LIN {X 0,Y 255.439,Z 401.538,A -85,B 0,C 180,E1 -18832.437,E2 -18832.437} C_VEL
LIN {X 0,Y 256.789,Z 390.953,A -85,B 0,C 180,E1 -18833.483,E2 -18833.483} C_VEL
LIN {X 0,Y 258.093,Z 377.272,A -85,B 0,C 180,E1 -18834.477,E2 -18834.477} C_VEL
LIN {X 0,Y 258.954,Z 364.44,A -85,B 0,C 180,E1 -18835.086,E2 -18835.086} C_VEL
LIN {X 0,Y 260.512,Z 307.195,A -85,B 0,C 180,E1 -18836.666,E2 -18836.666} C_VEL
LIN {X 0,Y 255.164,Z 263.56,A -85,B 0,C 180,E1 -18838.451,E2 -18838.451} C_VEL
LIN {X 0,Y 252.783,Z 256.222,A -85,B 0,C 180,E1 -18838.949,E2 -18838.949} C_VEL
LIN {X 0,Y 250.577,Z 245.438,A -85,B 0,C 180,E1 -18842.709,E2 -18842.709} C_VEL
LIN {X 0,Y 249.091,Z 238.46,A -85,B 0,C 180,E1 -18845.287,E2 -18845.287} C_VEL
LIN {X 0,Y 249.013,Z 238.47,A -85,B 0,C 180,E1 -18848.375,E2 -18848.375} C_VEL
LIN {X 0,Y 248.994,Z 238.467,A -85,B 0,C 180,E1 -18852.788,E2 -18852.788} C_VEL
LIN {X 0,Y 249.037,Z 238.464,A -85,B 0,C 180,E1 -18857.367,E2 -18857.367} C_VEL
LIN {X 0,Y 249.028,Z 238.466,A -85,B 0,C 180,E1 -18861.619,E2 -18861.619} C_VEL
LIN {X 0,Y 249.021,Z 238.467,A -85,B 0,C 180,E1 -18865.635,E2 -18865.635} C_VEL
LIN {X 0,Y 249.024,Z 238.466,A -85,B 0,C 180,E1 -18869.469,E2 -18869.469} C_VEL
LIN {X 0,Y 249.046,Z 238.462,A -85,B 0,C 180,E1 -18873.158,E2 -18873.158} C_VEL
LIN {X 0,Y 249.059,Z 238.457,A -85,B 0,C 180,E1 -18876.73,E2 -18876.73} C_VEL
LIN {X 0,Y 249.112,Z 238.451,A -85,B 0,C 180,E1 -18880.211,E2 -18880.211} C_VEL
LIN {X 0,Y 249.164,Z 238.448,A -85,B 0,C 180,E1 -18883.616,E2 -18883.616} C_VEL
LIN {X 0,Y 249.208,Z 238.435,A -85,B 0,C 180,E1 -18888.614,E2 -18888.614} C_VEL
LIN {X 0,Y 249.446,Z 238.411,A -85,B 0,C 180,E1 -18891.901,E2 -18891.901} C_VEL
LIN {X 0,Y 249.393,Z 238.406,A -85,B 0,C 180,E1 -18896.769,E2 -18896.769} C_VEL
LIN {X 0,Y 249.681,Z 238.355,A -85,B 0,C 180,E1 -18899.999,E2 -18899.999} C_VEL
LIN {X 0,Y 249.388,Z 238.41,A -85,B 0,C 180,E1 -18903.231,E2 -18903.231} C_VEL
LIN {X 0,Y 249.394,Z 238.415,A -85,B 0,C 180,E1 -18906.789,E2 -18906.789} C_VEL
LIN {X 0,Y 249.299,Z 238.426,A -85,B 0,C 180,E1 -18909.738,E2 -18909.738} C_VEL
LIN {X 0,Y 249.134,Z 238.452,A -85,B 0,C 180,E1 -18914.707,E2 -18914.707} C_VEL
LIN {X 0,Y 249.059,Z 238.457,A -85,B 0,C 180,E1 -18918.083,E2 -18918.083} C_VEL
LIN {X 0,Y 249.013,Z 238.463,A -85,B 0,C 180,E1 -18921.524,E2 -18921.524} C_VEL
LIN {X 0,Y 249.082,Z 238.453,A -85,B 0,C 180,E1 -18925.476,E2 -18925.476} C_VEL
LIN {X 0,Y 249.023,Z 238.445,A -85,B 0,C 180,E1 -18928.983,E2 -18928.983} C_VEL
LIN {X 0,Y 248.998,Z 238.45,A -85,B 0,C 180,E1 -18932.43,E2 -18932.43} C_VEL
LIN {X 0,Y 249.02,Z 238.465,A -85,B 0,C 180,E1 -18936.346,E2 -18936.346} C_VEL
LIN {X 0,Y 248.967,Z 238.464,A -85,B 0,C 180,E1 -18940.485,E2 -18940.485} C_VEL
LIN {X 0,Y 248.977,Z 238.453,A -85,B 0,C 180,E1 -18942.794,E2 -18942.794} C_VEL
LIN {X 0,Y 248.988,Z 238.468,A -85,B 0,C 180,E1 -18947.366,E2 -18947.366} C_VEL
LIN {X 0,Y 249.025,Z 238.455,A -85,B 0,C 180,E1 -18952.205,E2 -18952.205} C_VEL
LIN {X 0,Y 249.028,Z 238.464,A -85,B 0,C 180,E1 -18955.644,E2 -18955.644} C_VEL
LIN {X 0,Y 249.033,Z 238.457,A -85,B 0,C 180,E1 -18959.477,E2 -18959.477} C_VEL
LIN {X 0,Y 249.056,Z 238.46,A -85,B 0,C 180,E1 -18963.166,E2 -18963.166} C_VEL
LIN {X 0,Y 249.05,Z 238.461,A -85,B 0,C 180,E1 -18966.735,E2 -18966.735} C_VEL
LIN {X 0,Y 249.073,Z 238.462,A -85,B 0,C 180,E1 -18970.213,E2 -18970.213} C_VEL
LIN {X 0,Y 249.189,Z 238.45,A -85,B 0,C 180,E1 -18973.623,E2 -18973.623} C_VEL
LIN {X 0,Y 249.19,Z 238.451,A -85,B 0,C 180,E1 -18975.908,E2 -18975.908} C_VEL
LIN {X 0,Y 250.326,Z 241.478,A -85,B 0,C 180,E1 -18976.126,E2 -18976.126} C_VEL
LIN {X 0,Y 257.039,Z 256.974,A -85,B 0,C 180,E1 -18977.261,E2 -18977.261} C_VEL
LIN {X 0,Y 261.575,Z 270.407,A -85,B 0,C 180,E1 -18978.077,E2 -18978.077} C_VEL
LIN {X 0,Y 259.215,Z 342.899,A -85,B 0,C 180,E1 -18980.048,E2 -18980.048} C_VEL
LIN {X 0,Y 258.535,Z 356.06,A -85,B 0,C 180,E1 -18980.715,E2 -18980.715} C_VEL
LIN {X 0,Y 257.47,Z 368.762,A -85,B 0,C 180,E1 -18981.666,E2 -18981.666} C_VEL
LIN {X 0,Y 256.168,Z 380.863,A -85,B 0,C 180,E1 -18982.912,E2 -18982.912} C_VEL
LIN {X 0,Y 254.83,Z 392.116,A -85,B 0,C 180,E1 -18984.429,E2 -18984.429} C_VEL
LIN {X 0,Y 253.272,Z 402.421,A -85,B 0,C 180,E1 -18986.165,E2 -18986.165} C_VEL
LIN {X 0,Y 251.828,Z 411.246,A -85,B 0,C 180,E1 -18988.004,E2 -18988.004} C_VEL
LIN {X 0,Y 250.326,Z 420.436,A -85,B 0,C 180,E1 -18990.405,E2 -18990.405} C_VEL
LIN {X 0,Y 249.109,Z 427.844,A -85,B 0,C 180,E1 -18992.832,E2 -18992.832} C_VEL
LIN {X 0,Y 248.344,Z 432.864,A -85,B 0,C 180,E1 -18994.873,E2 -18994.873} C_VEL
LIN {X 0,Y 247.817,Z 437.113,A -85,B 0,C 180,E1 -18996.985,E2 -18996.985} C_VEL
LIN {X 0,Y 247.217,Z 441.489,A -85,B 0,C 180,E1 -18999.823,E2 -18999.823} C_VEL
LIN {X 0,Y 246.964,Z 443.438,A -85,B 0,C 180,E1 -19001.492,E2 -19001.492} C_VEL
LIN {X 0,Y 246.843,Z 445.788,A -85,B 0,C 180,E1 -19004.528,E2 -19004.528} C_VEL
LIN {X 0,Y 246.862,Z 446.599,A -85,B 0,C 180,E1 -19006.542,E2 -19006.542} C_VEL
LIN {X 0,Y 247.056,Z 446.823,A -85,B 0,C 180,E1 -19008.236,E2 -19008.236} C_VEL
LIN {X 0,Y 247.456,Z 446.467,A -85,B 0,C 180,E1 -19010.41,E2 -19010.41} C_VEL
LIN {X 0,Y 248.319,Z 444.912,A -85,B 0,C 180,E1 -19013.344,E2 -19013.344} C_VEL
LIN {X 0,Y 249.244,Z 442.844,A -85,B 0,C 180,E1 -19015.537,E2 -19015.537} C_VEL
LIN {X 0,Y 250.877,Z 438.906,A -85,B 0,C 180,E1 -19018.44,E2 -19018.44} C_VEL
LIN {X 0,Y 252.748,Z 434.14,A -85,B 0,C 180,E1 -19020.958,E2 -19020.958} C_VEL
LIN {X 0,Y 254.976,Z 427.989,A -85,B 0,C 180,E1 -19023.454,E2 -19023.454} C_VEL
LIN {X 0,Y 257.689,Z 420.236,A -85,B 0,C 180,E1 -19025.9,E2 -19025.9} C_VEL
LIN {X 0,Y 260.217,Z 412.22,A -85,B 0,C 180,E1 -19027.91,E2 -19027.91} C_VEL
LIN {X 0,Y 263.021,Z 402.281,A -85,B 0,C 180,E1 -19029.887,E2 -19029.887} C_VEL
LIN {X 0,Y 265.849,Z 391.372,A -85,B 0,C 180,E1 -19031.58,E2 -19031.58} C_VEL
LIN {X 0,Y 268.172,Z 380.195,A -85,B 0,C 180,E1 -19032.951,E2 -19032.951} C_VEL
LIN {X 0,Y 270.145,Z 367.926,A -85,B 0,C 180,E1 -19034.099,E2 -19034.099} C_VEL
LIN {X 0,Y 271.693,Z 355.388,A -85,B 0,C 180,E1 -19034.95,E2 -19034.95} C_VEL
LIN {X 0,Y 272.704,Z 342.7,A -85,B 0,C 180,E1 -19035.523,E2 -19035.523} C_VEL
LIN {X 0,Y 275.249,Z 284.695,A -85,B 0,C 180,E1 -19037.046,E2 -19037.046} C_VEL
LIN {X 0,Y 268.843,Z 271.231,A -85,B 0,C 180,E1 -19038.57,E2 -19038.57} C_VEL
LIN {X 0,Y 262.355,Z 259.216,A -85,B 0,C 180,E1 -19040.176,E2 -19040.176} C_VEL
LIN {X 0,Y 256.72,Z 250.714,A -85,B 0,C 180,E1 -19041.604,E2 -19041.604} C_VEL
LIN {X 0,Y 254.038,Z 246.769,A -85,B 0,C 180,E1 -19042.316,E2 -19042.316} C_VEL
LIN {X 0,Y 251.753,Z 243.157,A -85,B 0,C 180,E1 -19042.95,E2 -19042.95} C_VEL
LIN {X 0,Y 249.857,Z 240.911,A -85,B 0,C 180,E1 -19043.461,E2 -19043.461} C_VEL
LIN {X 0,Y 249.066,Z 238.461,A -85,B 0,C 180,E1 -19043.749,E2 -19043.749} C_VEL
LIN {X 0,Y 249.03,Z 238.456,A -85,B 0,C 180,E1 -19047.845,E2 -19047.845} C_VEL
LIN {X 0,Y 249.077,Z 238.447,A -85,B 0,C 180,E1 -19051.336,E2 -19051.336} C_VEL
LIN {X 0,Y 249.142,Z 238.437,A -85,B 0,C 180,E1 -19054.968,E2 -19054.968} C_VEL
LIN {X 0,Y 249.099,Z 238.45,A -85,B 0,C 180,E1 -19060.211,E2 -19060.211} C_VEL
LIN {X 0,Y 249.194,Z 238.434,A -85,B 0,C 180,E1 -19063.619,E2 -19063.619} C_VEL
LIN {X 0,Y 249.222,Z 238.435,A -85,B 0,C 180,E1 -19068.616,E2 -19068.616} C_VEL
LIN {X 0,Y 249.434,Z 238.4,A -85,B 0,C 180,E1 -19071.902,E2 -19071.902} C_VEL
LIN {X 0,Y 249.272,Z 238.426,A -85,B 0,C 180,E1 -19075.149,E2 -19075.149} C_VEL
LIN {X 0,Y 249.658,Z 238.38,A -85,B 0,C 180,E1 -19078.387,E2 -19078.387} C_VEL
LIN {X 0,Y 249.65,Z 238.369,A -85,B 0,C 180,E1 -19081.322,E2 -19081.322} C_VEL
LIN {X 0,Y 248.99,Z 238.46,A -85,B 0,C 180,E1 -19082.664,E2 -19082.664} C_VEL
LIN {X 0,Y 246.087,Z 238.832,A -85,B 0,C 180,E1 -19084.85,E2 -19084.85} C_VEL
LIN {X 0,Y 243.578,Z 239.148,A -85,B 0,C 180,E1 -19086.631,E2 -19086.631} C_VEL
LIN {X 0,Y 242.459,Z 239.28,A -85,B 0,C 180,E1 -19088.014,E2 -19088.014} C_VEL
LIN {X 0,Y 242.346,Z 239.289,A -85,B 0,C 180,E1 -19088.484,E2 -19088.484} C_VEL
LIN {X 0,Y 242.12,Z 239.317,A -85,B 0,C 180,E1 -19093.428,E2 -19093.428} C_VEL
LIN {X 0,Y 242.093,Z 239.326,A -85,B 0,C 180,E1 -19096.877,E2 -19096.877} C_VEL
LIN {X 0,Y 241.972,Z 239.339,A -85,B 0,C 180,E1 -19102.184,E2 -19102.184} C_VEL
LIN {X 0,Y 242.026,Z 239.337,A -85,B 0,C 180,E1 -19105.822,E2 -19105.822} C_VEL
LIN {X 0,Y 241.96,Z 239.346,A -85,B 0,C 180,E1 -19109.59,E2 -19109.59} C_VEL
LIN {X 0,Y 241.963,Z 239.342,A -85,B 0,C 180,E1 -19113.496,E2 -19113.496} C_VEL
LIN {X 0,Y 241.98,Z 239.336,A -85,B 0,C 180,E1 -19117.584,E2 -19117.584} C_VEL
LIN {X 0,Y 241.924,Z 239.326,A -85,B 0,C 180,E1 -19121.926,E2 -19121.926} C_VEL
LIN {X 0,Y 241.981,Z 239.548,A -85,B 0,C 180,E1 -19123.291,E2 -19123.291} C_VEL
LIN {X 0,Y 244.202,Z 246.816,A -85,B 0,C 180,E1 -19127.212,E2 -19127.212} C_VEL
LIN {X 0,Y 246.291,Z 254.002,A -85,B 0,C 180,E1 -19130.671,E2 -19130.671} C_VEL
LIN {X 0,Y 249.147,Z 258.875,A -85,B 0,C 180,E1 -19131.514,E2 -19131.514} C_VEL
LIN {X 0,Y 255.372,Z 270.327,A -85,B 0,C 180,E1 -19133.278,E2 -19133.278} C_VEL
LIN {X 0,Y 261.811,Z 283.473,A -85,B 0,C 180,E1 -19135.011,E2 -19135.011} C_VEL
LIN {X 0,Y 265.059,Z 291.167,A -85,B 0,C 180,E1 -19135.87,E2 -19135.87} C_VEL
LIN {X 0,Y 268.477,Z 313.345,A -85,B 0,C 180,E1 -19137.216,E2 -19137.216} C_VEL
LIN {X 0,Y 266.163,Z 364.461,A -85,B 0,C 180,E1 -19138.609,E2 -19138.609} C_VEL
LIN {X 0,Y 264.74,Z 377.806,A -85,B 0,C 180,E1 -19139.228,E2 -19139.228} C_VEL
LIN {X 0,Y 262.748,Z 390.649,A -85,B 0,C 180,E1 -19140.12,E2 -19140.12} C_VEL
LIN {X 0,Y 260.478,Z 401.692,A -85,B 0,C 180,E1 -19141.165,E2 -19141.165} C_VEL
LIN {X 0,Y 257.609,Z 413.215,A -85,B 0,C 180,E1 -19142.588,E2 -19142.588} C_VEL
LIN {X 0,Y 254.685,Z 423.609,A -85,B 0,C 180,E1 -19144.238,E2 -19144.238} C_VEL
LIN {X 0,Y 251.769,Z 433.003,A -85,B 0,C 180,E1 -19146.123,E2 -19146.123} C_VEL
LIN {X 0,Y 248.699,Z 442.088,A -85,B 0,C 180,E1 -19148.446,E2 -19148.446} C_VEL
LIN {X 0,Y 246.223,Z 449.442,A -85,B 0,C 180,E1 -19150.836,E2 -19150.836} C_VEL
LIN {X 0,Y 244.09,Z 455.377,A -85,B 0,C 180,E1 -19153.265,E2 -19153.265} C_VEL
LIN {X 0,Y 242.298,Z 460.092,A -85,B 0,C 180,E1 -19155.725,E2 -19155.725} C_VEL
LIN {X 0,Y 241.137,Z 463.725,A -85,B 0,C 180,E1 -19158.226,E2 -19158.226} C_VEL
LIN {X 0,Y 240.576,Z 465.619,A -85,B 0,C 180,E1 -19159.903,E2 -19159.903} C_VEL
LIN {X 0,Y 239.903,Z 468.104,A -85,B 0,C 180,E1 -19163.268,E2 -19163.268} C_VEL
LIN {X 0,Y 239.849,Z 468.8,A -85,B 0,C 180,E1 -19165.049,E2 -19165.049} C_VEL
LIN {X 0,Y 239.881,Z 469.054,A -85,B 0,C 180,E1 -19166.638,E2 -19166.638} C_VEL
LIN {X 0,Y 239.976,Z 468.912,A -85,B 0,C 180,E1 -19168.319,E2 -19168.319} C_VEL
LIN {X 0,Y 240.024,Z 468.36,A -85,B 0,C 180,E1 -19169.997,E2 -19169.997} C_VEL
LIN {X 0,Y 240.008,Z 467.408,A -85,B 0,C 180,E1 -19171.675,E2 -19171.675} C_VEL
LIN {X 0,Y 239.963,Z 466.048,A -85,B 0,C 180,E1 -19173.355,E2 -19173.355} C_VEL
LIN {X 0,Y 239.964,Z 463.14,A -85,B 0,C 180,E1 -19175.879,E2 -19175.879} C_VEL
LIN {X 0,Y 240.191,Z 459.169,A -85,B 0,C 180,E1 -19178.409,E2 -19178.409} C_VEL
LIN {X 0,Y 240.757,Z 453.024,A -85,B 0,C 180,E1 -19181.36,E2 -19181.36} C_VEL
LIN {X 0,Y 241.717,Z 446.284,A -85,B 0,C 180,E1 -19183.875,E2 -19183.875} C_VEL
LIN {X 0,Y 243.073,Z 437.902,A -85,B 0,C 180,E1 -19186.369,E2 -19186.369} C_VEL
LIN {X 0,Y 244.393,Z 429.258,A -85,B 0,C 180,E1 -19188.436,E2 -19188.436} C_VEL
LIN {X 0,Y 245.963,Z 419.772,A -85,B 0,C 180,E1 -19190.266,E2 -19190.266} C_VEL
LIN {X 0,Y 247.529,Z 409.43,A -85,B 0,C 180,E1 -19191.874,E2 -19191.874} C_VEL
LIN {X 0,Y 249.152,Z 398.134,A -85,B 0,C 180,E1 -19193.255,E2 -19193.255} C_VEL
LIN {X 0,Y 250.64,Z 385.426,A -85,B 0,C 180,E1 -19194.425,E2 -19194.425} C_VEL
LIN {X 0,Y 251.846,Z 371.806,A -85,B 0,C 180,E1 -19195.291,E2 -19195.291} C_VEL
LIN {X 0,Y 252.465,Z 359.698,A -85,B 0,C 180,E1 -19195.777,E2 -19195.777} C_VEL
LIN {X 0,Y 253.92,Z 308.786,A -85,B 0,C 180,E1 -19197.194,E2 -19197.194} C_VEL
LIN {X 0,Y 248.987,Z 266.806,A -85,B 0,C 180,E1 -19198.952,E2 -19198.952} C_VEL
LIN {X 0,Y 247.974,Z 262.879,A -85,B 0,C 180,E1 -19199.176,E2 -19199.176} C_VEL
LIN {X 0,Y 245.566,Z 256.004,A -85,B 0,C 180,E1 -19199.648,E2 -19199.648} C_VEL
LIN {X 0,Y 243.171,Z 244.542,A -85,B 0,C 180,E1 -19203.797,E2 -19203.797} C_VEL
LIN {X 0,Y 242.034,Z 239.342,A -85,B 0,C 180,E1 -19205.796,E2 -19205.796} C_VEL
LIN {X 0,Y 241.941,Z 239.35,A -85,B 0,C 180,E1 -19209.714,E2 -19209.714} C_VEL
LIN {X 0,Y 241.919,Z 239.35,A -85,B 0,C 180,E1 -19214.196,E2 -19214.196} C_VEL
LIN {X 0,Y 241.961,Z 239.346,A -85,B 0,C 180,E1 -19218.082,E2 -19218.082} C_VEL
LIN {X 0,Y 241.985,Z 239.34,A -85,B 0,C 180,E1 -19222.417,E2 -19222.417} C_VEL
LIN {X 0,Y 241.957,Z 239.342,A -85,B 0,C 180,E1 -19226.503,E2 -19226.503} C_VEL
LIN {X 0,Y 242.01,Z 239.335,A -85,B 0,C 180,E1 -19230.584,E2 -19230.584} C_VEL
LIN {X 0,Y 242.04,Z 239.333,A -85,B 0,C 180,E1 -19234.179,E2 -19234.179} C_VEL
LIN {X 0,Y 242.055,Z 239.332,A -85,B 0,C 180,E1 -19238.275,E2 -19238.275} C_VEL
LIN {X 0,Y 242.124,Z 239.323,A -85,B 0,C 180,E1 -19243.282,E2 -19243.282} C_VEL
LIN {X 0,Y 242.139,Z 239.315,A -85,B 0,C 180,E1 -19248.277,E2 -19248.277} C_VEL
LIN {X 0,Y 242.393,Z 239.291,A -85,B 0,C 180,E1 -19251.664,E2 -19251.664} C_VEL
LIN {X 0,Y 242.219,Z 239.307,A -85,B 0,C 180,E1 -19255.006,E2 -19255.006} C_VEL
LIN {X 0,Y 242.597,Z 239.242,A -85,B 0,C 180,E1 -19258.339,E2 -19258.339} C_VEL
LIN {X 0,Y 242.595,Z 239.247,A -85,B 0,C 180,E1 -19261.66,E2 -19261.66} C_VEL
LIN {X 0,Y 242.373,Z 239.292,A -85,B 0,C 180,E1 -19266.762,E2 -19266.762} C_VEL
LIN {X 0,Y 242.228,Z 239.306,A -85,B 0,C 180,E1 -19270.025,E2 -19270.025} C_VEL
LIN {X 0,Y 242.086,Z 239.33,A -85,B 0,C 180,E1 -19275.145,E2 -19275.145} C_VEL
LIN {X 0,Y 241.996,Z 239.335,A -85,B 0,C 180,E1 -19278.63,E2 -19278.63} C_VEL
LIN {X 0,Y 241.956,Z 239.343,A -85,B 0,C 180,E1 -19282.185,E2 -19282.185} C_VEL
LIN {X 0,Y 242.02,Z 239.333,A -85,B 0,C 180,E1 -19285.832,E2 -19285.832} C_VEL
LIN {X 0,Y 241.946,Z 239.324,A -85,B 0,C 180,E1 -19289.591,E2 -19289.591} C_VEL
LIN {X 0,Y 241.951,Z 239.335,A -85,B 0,C 180,E1 -19293.497,E2 -19293.497} C_VEL
LIN {X 0,Y 241.962,Z 239.342,A -85,B 0,C 180,E1 -19297.586,E2 -19297.586} C_VEL
LIN {X 0,Y 241.906,Z 239.337,A -85,B 0,C 180,E1 -19301.928,E2 -19301.928} C_VEL
LIN {X 0,Y 241.904,Z 239.352,A -85,B 0,C 180,E1 -19306.578,E2 -19306.578} C_VEL
LIN {X 0,Y 241.977,Z 239.334,A -85,B 0,C 180,E1 -19311.645,E2 -19311.645} C_VEL
LIN {X 0,Y 241.964,Z 239.343,A -85,B 0,C 180,E1 -19314.493,E2 -19314.493} C_VEL
LIN {X 0,Y 241.958,Z 239.339,A -85,B 0,C 180,E1 -19318.484,E2 -19318.484} C_VEL
LIN {X 0,Y 241.989,Z 239.343,A -85,B 0,C 180,E1 -19322.316,E2 -19322.316} C_VEL
LIN {X 0,Y 242.03,Z 239.337,A -85,B 0,C 180,E1 -19326.019,E2 -19326.019} C_VEL
LIN {X 0,Y 242.01,Z 239.341,A -85,B 0,C 180,E1 -19329.611,E2 -19329.611} C_VEL
LIN {X 0,Y 242.109,Z 239.332,A -85,B 0,C 180,E1 -19333.32,E2 -19333.32} C_VEL
LIN {X 0,Y 242.154,Z 239.407,A -85,B 0,C 180,E1 -19335.201,E2 -19335.201} C_VEL
LIN {X 0,Y 243.167,Z 242.232,A -85,B 0,C 180,E1 -19335.402,E2 -19335.402} C_VEL
LIN {X 0,Y 250.184,Z 257.809,A -85,B 0,C 180,E1 -19336.62,E2 -19336.62} C_VEL
LIN {X 0,Y 254.989,Z 271.769,A -85,B 0,C 180,E1 -19337.515,E2 -19337.515} C_VEL
LIN {X 0,Y 252.534,Z 343.875,A -85,B 0,C 180,E1 -19339.531,E2 -19339.531} C_VEL
LIN {X 0,Y 251.772,Z 357.541,A -85,B 0,C 180,E1 -19340.261,E2 -19340.261} C_VEL
LIN {X 0,Y 250.666,Z 369.927,A -85,B 0,C 180,E1 -19341.235,E2 -19341.235} C_VEL
LIN {X 0,Y 249.317,Z 381.794,A -85,B 0,C 180,E1 -19342.512,E2 -19342.512} C_VEL
LIN {X 0,Y 247.812,Z 393.628,A -85,B 0,C 180,E1 -19344.175,E2 -19344.175} C_VEL
LIN {X 0,Y 246.155,Z 404.168,A -85,B 0,C 180,E1 -19346.054,E2 -19346.054} C_VEL
LIN {X 0,Y 244.419,Z 414.357,A -85,B 0,C 180,E1 -19348.355,E2 -19348.355} C_VEL
LIN {X 0,Y 243.176,Z 421.706,A -85,B 0,C 180,E1 -19350.417,E2 -19350.417} C_VEL
LIN {X 0,Y 241.98,Z 428.94,A -85,B 0,C 180,E1 -19352.916,E2 -19352.916} C_VEL
LIN {X 0,Y 241.206,Z 433.823,A -85,B 0,C 180,E1 -19355.017,E2 -19355.017} C_VEL
LIN {X 0,Y 240.569,Z 438.563,A -85,B 0,C 180,E1 -19357.556,E2 -19357.556} C_VEL
LIN {X 0,Y 240.056,Z 442.199,A -85,B 0,C 180,E1 -19360.119,E2 -19360.119} C_VEL
LIN {X 0,Y 239.843,Z 444.046,A -85,B 0,C 180,E1 -19361.838,E2 -19361.838} C_VEL
LIN {X 0,Y 239.753,Z 446.126,A -85,B 0,C 180,E1 -19364.685,E2 -19364.685} C_VEL
LIN {X 0,Y 239.821,Z 447.01,A -85,B 0,C 180,E1 -19367.042,E2 -19367.042} C_VEL
LIN {X 0,Y 240.053,Z 447.131,A -85,B 0,C 180,E1 -19368.788,E2 -19368.788} C_VEL
LIN {X 0,Y 240.439,Z 446.8,A -85,B 0,C 180,E1 -19370.716,E2 -19370.716} C_VEL
LIN {X 0,Y 240.88,Z 446.156,A -85,B 0,C 180,E1 -19372.291,E2 -19372.291} C_VEL
LIN {X 0,Y 241.471,Z 444.998,A -85,B 0,C 180,E1 -19374.047,E2 -19374.047} C_VEL
LIN {X 0,Y 242.342,Z 443.2,A -85,B 0,C 180,E1 -19375.973,E2 -19375.973} C_VEL
LIN {X 0,Y 243.732,Z 440.081,A -85,B 0,C 180,E1 -19378.41,E2 -19378.41} C_VEL
LIN {X 0,Y 245.62,Z 435.601,A -85,B 0,C 180,E1 -19381,E2 -19381} C_VEL
LIN {X 0,Y 247.883,Z 429.807,A -85,B 0,C 180,E1 -19383.564,E2 -19383.564} C_VEL
LIN {X 0,Y 250.653,Z 422.421,A -85,B 0,C 180,E1 -19386.073,E2 -19386.073} C_VEL
LIN {X 0,Y 253.201,Z 414.791,A -85,B 0,C 180,E1 -19388.139,E2 -19388.139} C_VEL
LIN {X 0,Y 256.282,Z 404.734,A -85,B 0,C 180,E1 -19390.303,E2 -19390.303} C_VEL
LIN {X 0,Y 259.021,Z 395.064,A -85,B 0,C 180,E1 -19391.923,E2 -19391.923} C_VEL
LIN {X 0,Y 261.61,Z 383.714,A -85,B 0,C 180,E1 -19393.436,E2 -19393.436} C_VEL
LIN {X 0,Y 263.736,Z 371.991,A -85,B 0,C 180,E1 -19394.653,E2 -19394.653} C_VEL
LIN {X 0,Y 265.523,Z 359.394,A -85,B 0,C 180,E1 -19395.613,E2 -19395.613} C_VEL
LIN {X 0,Y 266.799,Z 346.003,A -85,B 0,C 180,E1 -19396.297,E2 -19396.297} C_VEL
LIN {X 0,Y 268.025,Z 322.583,A -85,B 0,C 180,E1 -19396.962,E2 -19396.962} C_VEL
LIN {X 0,Y 269.62,Z 286.994,A -85,B 0,C 180,E1 -19397.899,E2 -19397.899} C_VEL
LIN {X 0,Y 262.712,Z 272.581,A -85,B 0,C 180,E1 -19399.628,E2 -19399.628} C_VEL
LIN {X 0,Y 256.927,Z 262.324,A -85,B 0,C 180,E1 -19401.124,E2 -19401.124} C_VEL
LIN {X 0,Y 250.399,Z 252.33,A -85,B 0,C 180,E1 -19402.884,E2 -19402.884} C_VEL
LIN {X 0,Y 247.34,Z 247.994,A -85,B 0,C 180,E1 -19403.746,E2 -19403.746} C_VEL
LIN {X 0,Y 245.179,Z 244.537,A -85,B 0,C 180,E1 -19404.395,E2 -19404.395} C_VEL
LIN {X 0,Y 242.833,Z 241.862,A -85,B 0,C 180,E1 -19405.076,E2 -19405.076} C_VEL
LIN {X 0,Y 242.014,Z 239.331,A -85,B 0,C 180,E1 -19405.415,E2 -19405.415} C_VEL
LIN {X 0,Y 241.999,Z 239.334,A -85,B 0,C 180,E1 -19410.416,E2 -19410.416} C_VEL
LIN {X 0,Y 242.06,Z 239.323,A -85,B 0,C 180,E1 -19414.183,E2 -19414.183} C_VEL
LIN {X 0,Y 242.044,Z 239.323,A -85,B 0,C 180,E1 -19418.298,E2 -19418.298} C_VEL
LIN {X 0,Y 242.154,Z 239.309,A -85,B 0,C 180,E1 -19423.278,E2 -19423.278} C_VEL
LIN {X 0,Y 242.157,Z 239.312,A -85,B 0,C 180,E1 -19428.279,E2 -19428.279} C_VEL
LIN {X 0,Y 242.381,Z 239.279,A -85,B 0,C 180,E1 -19431.665,E2 -19431.665} C_VEL
LIN {X 0,Y 242.405,Z 239.282,A -85,B 0,C 180,E1 -19433.341,E2 -19433.341} C_VEL
LIN {X 0,Y 242.619,Z 239.257,A -85,B 0,C 180,E1 -19438.341,E2 -19438.341} C_VEL
LIN {X 0,Y 242.618,Z 239.246,A -85,B 0,C 180,E1 -19441.66,E2 -19441.66} C_VEL
LIN {X 0,Y 242.385,Z 239.276,A -85,B 0,C 180,E1 -19446.661,E2 -19446.661} C_VEL
LIN {X 0,Y 242.346,Z 239.289,A -85,B 0,C 180,E1 -19448.484,E2 -19448.484} C_VEL
LIN {X 0,Y 241.606,Z 239.374,A -85,B 0,C 180,E1 -19449.868,E2 -19449.868} C_VEL
LIN {X 0,Y 238.682,Z 239.747,A -85,B 0,C 180,E1 -19452.123,E2 -19452.123} C_VEL
LIN {X 0,Y 236.219,Z 240.049,A -85,B 0,C 180,E1 -19453.96,E2 -19453.96} C_VEL
LIN {X 0,Y 235.146,Z 240.181,A -85,B 0,C 180,E1 -19455.388,E2 -19455.388} C_VEL
LIN {X 0,Y 235.047,Z 240.194,A -85,B 0,C 180,E1 -19455.872,E2 -19455.872} C_VEL
LIN {X 0,Y 234.93,Z 240.22,A -85,B 0,C 180,E1 -19461.038,E2 -19461.038} C_VEL
LIN {X 0,Y 234.962,Z 240.213,A -85,B 0,C 180,E1 -19466.194,E2 -19466.194} C_VEL
LIN {X 0,Y 234.883,Z 240.219,A -85,B 0,C 180,E1 -19470.575,E2 -19470.575} C_VEL
LIN {X 0,Y 234.894,Z 240.218,A -85,B 0,C 180,E1 -19474.645,E2 -19474.645} C_VEL
LIN {X 0,Y 234.91,Z 240.225,A -85,B 0,C 180,E1 -19478.936,E2 -19478.936} C_VEL
LIN {X 0,Y 234.894,Z 240.225,A -85,B 0,C 180,E1 -19481.584,E2 -19481.584} C_VEL
LIN {X 0,Y 237.287,Z 247.923,A -85,B 0,C 180,E1 -19486.02,E2 -19486.02} C_VEL
LIN {X 0,Y 238.935,Z 253.518,A -85,B 0,C 180,E1 -19488.863,E2 -19488.863} C_VEL
LIN {X 0,Y 241.712,Z 258.238,A -85,B 0,C 180,E1 -19489.762,E2 -19489.762} C_VEL
LIN {X 0,Y 246.409,Z 266.402,A -85,B 0,C 180,E1 -19491.204,E2 -19491.204} C_VEL
LIN {X 0,Y 251.242,Z 275.433,A -85,B 0,C 180,E1 -19492.619,E2 -19492.619} C_VEL
LIN {X 0,Y 257.32,Z 288.042,A -85,B 0,C 180,E1 -19494.325,E2 -19494.325} C_VEL
LIN {X 0,Y 259.874,Z 294.298,A -85,B 0,C 180,E1 -19495.039,E2 -19495.039} C_VEL
LIN {X 0,Y 262.897,Z 314.711,A -85,B 0,C 180,E1 -19496.311,E2 -19496.311} C_VEL
LIN {X 0,Y 260.482,Z 364.486,A -85,B 0,C 180,E1 -19497.686,E2 -19497.686} C_VEL
LIN {X 0,Y 258.965,Z 378.06,A -85,B 0,C 180,E1 -19498.334,E2 -19498.334} C_VEL
LIN {X 0,Y 257.054,Z 389.808,A -85,B 0,C 180,E1 -19499.16,E2 -19499.16} C_VEL
LIN {X 0,Y 254.693,Z 400.991,A -85,B 0,C 180,E1 -19500.218,E2 -19500.218} C_VEL
LIN {X 0,Y 251.697,Z 412.585,A -85,B 0,C 180,E1 -19501.661,E2 -19501.661} C_VEL
LIN {X 0,Y 248.623,Z 423.031,A -85,B 0,C 180,E1 -19503.336,E2 -19503.336} C_VEL
LIN {X 0,Y 245.876,Z 431.591,A -85,B 0,C 180,E1 -19505.063,E2 -19505.063} C_VEL
LIN {X 0,Y 243.106,Z 439.509,A -85,B 0,C 180,E1 -19507.028,E2 -19507.028} C_VEL
LIN {X 0,Y 240.321,Z 447.298,A -85,B 0,C 180,E1 -19509.455,E2 -19509.455} C_VEL
LIN {X 0,Y 237.945,Z 453.566,A -85,B 0,C 180,E1 -19511.932,E2 -19511.932} C_VEL
LIN {X 0,Y 235.983,Z 458.587,A -85,B 0,C 180,E1 -19514.451,E2 -19514.451} C_VEL
LIN {X 0,Y 234.473,Z 462.505,A -85,B 0,C 180,E1 -19517.007,E2 -19517.007} C_VEL
LIN {X 0,Y 233.555,Z 465.429,A -85,B 0,C 180,E1 -19519.596,E2 -19519.596} C_VEL
LIN {X 0,Y 232.824,Z 467.848,A -85,B 0,C 180,E1 -19523.063,E2 -19523.063} C_VEL
LIN {X 0,Y 232.775,Z 468.566,A -85,B 0,C 180,E1 -19525.107,E2 -19525.107} C_VEL
LIN {X 0,Y 232.903,Z 468.54,A -85,B 0,C 180,E1 -19528.268,E2 -19528.268} C_VEL
LIN {X 0,Y 232.952,Z 467.96,A -85,B 0,C 180,E1 -19529.997,E2 -19529.997} C_VEL
LIN {X 0,Y 232.937,Z 466.979,A -85,B 0,C 180,E1 -19531.726,E2 -19531.726} C_VEL
LIN {X 0,Y 232.879,Z 465.575,A -85,B 0,C 180,E1 -19533.457,E2 -19533.457} C_VEL
LIN {X 0,Y 232.9,Z 462.612,A -85,B 0,C 180,E1 -19536.059,E2 -19536.059} C_VEL
LIN {X 0,Y 233.127,Z 458.573,A -85,B 0,C 180,E1 -19538.666,E2 -19538.666} C_VEL
LIN {X 0,Y 233.748,Z 452.322,A -85,B 0,C 180,E1 -19541.705,E2 -19541.705} C_VEL
LIN {X 0,Y 234.788,Z 445.5,A -85,B 0,C 180,E1 -19544.293,E2 -19544.293} C_VEL
LIN {X 0,Y 236.245,Z 437.008,A -85,B 0,C 180,E1 -19546.856,E2 -19546.856} C_VEL
LIN {X 0,Y 237.623,Z 428.208,A -85,B 0,C 180,E1 -19548.981,E2 -19548.981} C_VEL
LIN {X 0,Y 239.208,Z 418.564,A -85,B 0,C 180,E1 -19550.864,E2 -19550.864} C_VEL
LIN {X 0,Y 240.837,Z 408.031,A -85,B 0,C 180,E1 -19552.515,E2 -19552.515} C_VEL
LIN {X 0,Y 242.656,Z 396.499,A -85,B 0,C 180,E1 -19553.916,E2 -19553.916} C_VEL
LIN {X 0,Y 244.035,Z 384.492,A -85,B 0,C 180,E1 -19555.018,E2 -19555.018} C_VEL
LIN {X 0,Y 245.202,Z 371.54,A -85,B 0,C 180,E1 -19555.856,E2 -19555.856} C_VEL
LIN {X 0,Y 245.908,Z 357.828,A -85,B 0,C 180,E1 -19556.403,E2 -19556.403} C_VEL
LIN {X 0,Y 247.278,Z 308.652,A -85,B 0,C 180,E1 -19557.81,E2 -19557.81} C_VEL
LIN {X 0,Y 242.457,Z 267.665,A -85,B 0,C 180,E1 -19559.587,E2 -19559.587} C_VEL
LIN {X 0,Y 238.266,Z 255.572,A -85,B 0,C 180,E1 -19560.463,E2 -19560.463} C_VEL
LIN {X 0,Y 235.704,Z 243.521,A -85,B 0,C 180,E1 -19565.013,E2 -19565.013} C_VEL
LIN {X 0,Y 234.984,Z 240.219,A -85,B 0,C 180,E1 -19566.366,E2 -19566.366} C_VEL
LIN {X 0,Y 234.928,Z 240.224,A -85,B 0,C 180,E1 -19568.939,E2 -19568.939} C_VEL
LIN {X 0,Y 234.873,Z 240.228,A -85,B 0,C 180,E1 -19573.48,E2 -19573.48} C_VEL
LIN {X 0,Y 234.941,Z 240.219,A -85,B 0,C 180,E1 -19576.526,E2 -19576.526} C_VEL
LIN {X 0,Y 234.934,Z 240.218,A -85,B 0,C 180,E1 -19581.081,E2 -19581.081} C_VEL
LIN {X 0,Y 234.911,Z 240.223,A -85,B 0,C 180,E1 -19585.358,E2 -19585.358} C_VEL
LIN {X 0,Y 234.905,Z 240.225,A -85,B 0,C 180,E1 -19589.428,E2 -19589.428} C_VEL
LIN {X 0,Y 234.967,Z 240.216,A -85,B 0,C 180,E1 -19593.79,E2 -19593.79} C_VEL
LIN {X 0,Y 235.012,Z 240.211,A -85,B 0,C 180,E1 -19598.969,E2 -19598.969} C_VEL
LIN {X 0,Y 235.06,Z 240.201,A -85,B 0,C 180,E1 -19603.062,E2 -19603.062} C_VEL
LIN {X 0,Y 235.07,Z 240.196,A -85,B 0,C 180,E1 -19607.919,E2 -19607.919} C_VEL
LIN {X 0,Y 235.342,Z 240.17,A -85,B 0,C 180,E1 -19611.412,E2 -19611.412} C_VEL
LIN {X 0,Y 235.368,Z 240.166,A -85,B 0,C 180,E1 -19613.14,E2 -19613.14} C_VEL
LIN {X 0,Y 235.557,Z 240.117,A -85,B 0,C 180,E1 -19618.29,E2 -19618.29} C_VEL
LIN {X 0,Y 235.555,Z 240.123,A -85,B 0,C 180,E1 -19621.709,E2 -19621.709} C_VEL
LIN {X 0,Y 235.331,Z 240.171,A -85,B 0,C 180,E1 -19626.86,E2 -19626.86} C_VEL
LIN {X 0,Y 235.176,Z 240.185,A -85,B 0,C 180,E1 -19630.329,E2 -19630.329} C_VEL
LIN {X 0,Y 235.035,Z 240.206,A -85,B 0,C 180,E1 -19635.611,E2 -19635.611} C_VEL
LIN {X 0,Y 234.935,Z 240.212,A -85,B 0,C 180,E1 -19639.211,E2 -19639.211} C_VEL
LIN {X 0,Y 234.911,Z 240.224,A -85,B 0,C 180,E1 -19642.887,E2 -19642.887} C_VEL
LIN {X 0,Y 234.926,Z 240.213,A -85,B 0,C 180,E1 -19646.662,E2 -19646.662} C_VEL
LIN {X 0,Y 234.872,Z 240.199,A -85,B 0,C 180,E1 -19650.576,E2 -19650.576} C_VEL
LIN {X 0,Y 234.902,Z 240.218,A -85,B 0,C 180,E1 -19654.642,E2 -19654.642} C_VEL
LIN {X 0,Y 234.888,Z 240.222,A -85,B 0,C 180,E1 -19658.939,E2 -19658.939} C_VEL
LIN {X 0,Y 234.855,Z 240.21,A -85,B 0,C 180,E1 -19663.493,E2 -19663.493} C_VEL
LIN {X 0,Y 234.857,Z 240.229,A -85,B 0,C 180,E1 -19666.516,E2 -19666.516} C_VEL
LIN {X 0,Y 234.9,Z 240.216,A -85,B 0,C 180,E1 -19671.083,E2 -19671.083} C_VEL
LIN {X 0,Y 234.911,Z 240.221,A -85,B 0,C 180,E1 -19675.366,E2 -19675.366} C_VEL
LIN {X 0,Y 234.908,Z 240.215,A -85,B 0,C 180,E1 -19679.435,E2 -19679.435} C_VEL
LIN {X 0,Y 234.983,Z 240.215,A -85,B 0,C 180,E1 -19683.799,E2 -19683.799} C_VEL
LIN {X 0,Y 234.961,Z 240.217,A -85,B 0,C 180,E1 -19688.97,E2 -19688.97} C_VEL
LIN {X 0,Y 235.049,Z 240.211,A -85,B 0,C 180,E1 -19693.096,E2 -19693.096} C_VEL
LIN {X 0,Y 235.072,Z 240.209,A -85,B 0,C 180,E1 -19694.423,E2 -19694.423} C_VEL
LIN {X 0,Y 236.157,Z 243.161,A -85,B 0,C 180,E1 -19694.654,E2 -19694.654} C_VEL
LIN {X 0,Y 244.013,Z 260.374,A -85,B 0,C 180,E1 -19696.075,E2 -19696.075} C_VEL
LIN {X 0,Y 248.399,Z 273.131,A -85,B 0,C 180,E1 -19696.922,E2 -19696.922} C_VEL
LIN {X 0,Y 245.929,Z 343.671,A -85,B 0,C 180,E1 -19698.934,E2 -19698.934} C_VEL
LIN {X 0,Y 245.179,Z 356.76,A -85,B 0,C 180,E1 -19699.631,E2 -19699.631} C_VEL
LIN {X 0,Y 243.981,Z 370.004,A -85,B 0,C 180,E1 -19700.679,E2 -19700.679} C_VEL
LIN {X 0,Y 242.699,Z 381.138,A -85,B 0,C 180,E1 -19701.888,E2 -19701.888} C_VEL
LIN {X 0,Y 241.376,Z 391.399,A -85,B 0,C 180,E1 -19703.315,E2 -19703.315} C_VEL
LIN {X 0,Y 239.714,Z 402.059,A -85,B 0,C 180,E1 -19705.168,E2 -19705.168} C_VEL
LIN {X 0,Y 238.186,Z 410.787,A -85,B 0,C 180,E1 -19707.043,E2 -19707.043} C_VEL
LIN {X 0,Y 236.72,Z 418.821,A -85,B 0,C 180,E1 -19709.152,E2 -19709.152} C_VEL
LIN {X 0,Y 235.364,Z 426.671,A -85,B 0,C 180,E1 -19711.714,E2 -19711.714} C_VEL
LIN {X 0,Y 234.339,Z 432.948,A -85,B 0,C 180,E1 -19714.302,E2 -19714.302} C_VEL
LIN {X 0,Y 233.642,Z 438.01,A -85,B 0,C 180,E1 -19716.957,E2 -19716.957} C_VEL
LIN {X 0,Y 233.084,Z 441.807,A -85,B 0,C 180,E1 -19719.548,E2 -19719.548} C_VEL
LIN {X 0,Y 232.738,Z 444.634,A -85,B 0,C 180,E1 -19722.205,E2 -19722.205} C_VEL
LIN {X 0,Y 232.656,Z 446.461,A -85,B 0,C 180,E1 -19724.842,E2 -19724.842} C_VEL
LIN {X 0,Y 232.792,Z 447.378,A -85,B 0,C 180,E1 -19727.573,E2 -19727.573} C_VEL
LIN {X 0,Y 233.425,Z 447.134,A -85,B 0,C 180,E1 -19731.038,E2 -19731.038} C_VEL
LIN {X 0,Y 233.989,Z 446.319,A -85,B 0,C 180,E1 -19732.984,E2 -19732.984} C_VEL
LIN {X 0,Y 235.486,Z 443.542,A -85,B 0,C 180,E1 -19736.449,E2 -19736.449} C_VEL
LIN {X 0,Y 237.158,Z 439.977,A -85,B 0,C 180,E1 -19739.273,E2 -19739.273} C_VEL
LIN {X 0,Y 239.234,Z 435.366,A -85,B 0,C 180,E1 -19741.924,E2 -19741.924} C_VEL
LIN {X 0,Y 241.683,Z 429.382,A -85,B 0,C 180,E1 -19744.545,E2 -19744.545} C_VEL
LIN {X 0,Y 244.622,Z 421.794,A -85,B 0,C 180,E1 -19747.108,E2 -19747.108} C_VEL
LIN {X 0,Y 247.355,Z 413.981,A -85,B 0,C 180,E1 -19749.207,E2 -19749.207} C_VEL
LIN {X 0,Y 250.439,Z 404.386,A -85,B 0,C 180,E1 -19751.259,E2 -19751.259} C_VEL
LIN {X 0,Y 253.5,Z 393.562,A -85,B 0,C 180,E1 -19753.054,E2 -19753.054} C_VEL
LIN {X 0,Y 255.994,Z 382.9,A -85,B 0,C 180,E1 -19754.456,E2 -19754.456} C_VEL
LIN {X 0,Y 258.279,Z 370.47,A -85,B 0,C 180,E1 -19755.722,E2 -19755.722} C_VEL
LIN {X 0,Y 260.149,Z 356.996,A -85,B 0,C 180,E1 -19756.694,E2 -19756.694} C_VEL
LIN {X 0,Y 261.282,Z 344.726,A -85,B 0,C 180,E1 -19757.289,E2 -19757.289} C_VEL
LIN {X 0,Y 264.022,Z 289.43,A -85,B 0,C 180,E1 -19758.79,E2 -19758.79} C_VEL
LIN {X 0,Y 257.942,Z 276.58,A -85,B 0,C 180,E1 -19760.393,E2 -19760.393} C_VEL
LIN {X 0,Y 252.55,Z 266.901,A -85,B 0,C 180,E1 -19761.851,E2 -19761.851} C_VEL
LIN {X 0,Y 246.177,Z 257.11,A -85,B 0,C 180,E1 -19763.643,E2 -19763.643} C_VEL
LIN {X 0,Y 243.26,Z 252.911,A -85,B 0,C 180,E1 -19764.505,E2 -19764.505} C_VEL
LIN {X 0,Y 240.793,Z 249.306,A -85,B 0,C 180,E1 -19765.264,E2 -19765.264} C_VEL
LIN {X 0,Y 238.588,Z 246.142,A -85,B 0,C 180,E1 -19765.967,E2 -19765.967} C_VEL
LIN {X 0,Y 237.905,Z 245.147,A -85,B 0,C 180,E1 -19766.19,E2 -19766.19} C_VEL
LIN {X 0,Y 235.835,Z 242.9,A -85,B 0,C 180,E1 -19766.845,E2 -19766.845} C_VEL
LIN {X 0,Y 234.958,Z 240.212,A -85,B 0,C 180,E1 -19767.233,E2 -19767.233} C_VEL
LIN {X 0,Y 234.928,Z 240.209,A -85,B 0,C 180,E1 -19771.403,E2 -19771.403} C_VEL
LIN {X 0,Y 234.978,Z 240.201,A -85,B 0,C 180,E1 -19775.246,E2 -19775.246} C_VEL
LIN {X 0,Y 235.002,Z 240.198,A -85,B 0,C 180,E1 -19778.97,E2 -19778.97} C_VEL
LIN {X 0,Y 235.087,Z 240.189,A -85,B 0,C 180,E1 -19783.061,E2 -19783.061} C_VEL
LIN {X 0,Y 235.09,Z 240.19,A -85,B 0,C 180,E1 -19787.921,E2 -19787.921} C_VEL
LIN {X 0,Y 235.31,Z 240.161,A -85,B 0,C 180,E1 -19791.412,E2 -19791.412} C_VEL
LIN {X 0,Y 235.356,Z 240.159,A -85,B 0,C 180,E1 -19793.14,E2 -19793.14} C_VEL
LIN {X 0,Y 235.578,Z 240.134,A -85,B 0,C 180,E1 -19798.291,E2 -19798.291} C_VEL
LIN {X 0,Y 235.577,Z 240.123,A -85,B 0,C 180,E1 -19801.71,E2 -19801.71} C_VEL
LIN {X 0,Y 235.336,Z 240.155,A -85,B 0,C 180,E1 -19806.861,E2 -19806.861} C_VEL
LIN {X 0,Y 235.176,Z 240.171,A -85,B 0,C 180,E1 -19810.33,E2 -19810.33} C_VEL
LIN {X 0,Y 235.06,Z 240.192,A -85,B 0,C 180,E1 -19815.611,E2 -19815.611} C_VEL
LIN {X 0,Y 235.047,Z 240.194,A -85,B 0,C 180,E1 -19815.872,E2 -19815.872} C_VEL
LIN {X 0,Y 234.333,Z 240.292,A -85,B 0,C 180,E1 -19817.3,E2 -19817.3} C_VEL
LIN {X 0,Y 231.412,Z 240.652,A -85,B 0,C 180,E1 -19819.628,E2 -19819.628} C_VEL
LIN {X 0,Y 228.966,Z 240.963,A -85,B 0,C 180,E1 -19821.527,E2 -19821.527} C_VEL
LIN {X 0,Y 227.943,Z 241.081,A -85,B 0,C 180,E1 -19823.002,E2 -19823.002} C_VEL
LIN {X 0,Y 227.872,Z 241.089,A -85,B 0,C 180,E1 -19823.502,E2 -19823.502} C_VEL
LIN {X 0,Y 227.847,Z 241.093,A -85,B 0,C 180,E1 -19827.561,E2 -19827.561} C_VEL
LIN {X 0,Y 227.836,Z 241.097,A -85,B 0,C 180,E1 -19831.628,E2 -19831.628} C_VEL
LIN {X 0,Y 227.857,Z 241.102,A -85,B 0,C 180,E1 -19835.877,E2 -19835.877} C_VEL
LIN {X 0,Y 227.822,Z 241.236,A -85,B 0,C 180,E1 -19839.884,E2 -19839.884} C_VEL
LIN {X 0,Y 229.668,Z 246.993,A -85,B 0,C 180,E1 -19843.512,E2 -19843.512} C_VEL
LIN {X 0,Y 231.507,Z 252.949,A -85,B 0,C 180,E1 -19846.834,E2 -19846.834} C_VEL
LIN {X 0,Y 234.307,Z 257.608,A -85,B 0,C 180,E1 -19847.827,E2 -19847.827} C_VEL
LIN {X 0,Y 239.066,Z 265.495,A -85,B 0,C 180,E1 -19849.419,E2 -19849.419} C_VEL
LIN {X 0,Y 244.124,Z 274.53,A -85,B 0,C 180,E1 -19851.014,E2 -19851.014} C_VEL
LIN {X 0,Y 250.36,Z 287.024,A -85,B 0,C 180,E1 -19852.884,E2 -19852.884} C_VEL
LIN {X 0,Y 254.71,Z 297.184,A -85,B 0,C 180,E1 -19854.153,E2 -19854.153} C_VEL
LIN {X 0,Y 257.387,Z 315.712,A -85,B 0,C 180,E1 -19855.349,E2 -19855.349} C_VEL
LIN {X 0,Y 254.89,Z 364.282,A -85,B 0,C 180,E1 -19856.711,E2 -19856.711} C_VEL
LIN {X 0,Y 253.306,Z 377.808,A -85,B 0,C 180,E1 -19857.364,E2 -19857.364} C_VEL
LIN {X 0,Y 251.242,Z 390.062,A -85,B 0,C 180,E1 -19858.248,E2 -19858.248} C_VEL
LIN {X 0,Y 248.602,Z 401.864,A -85,B 0,C 180,E1 -19859.412,E2 -19859.412} C_VEL
LIN {X 0,Y 245.513,Z 413.236,A -85,B 0,C 180,E1 -19860.88,E2 -19860.88} C_VEL
LIN {X 0,Y 242.333,Z 423.515,A -85,B 0,C 180,E1 -19862.587,E2 -19862.587} C_VEL
LIN {X 0,Y 239.477,Z 431.939,A -85,B 0,C 180,E1 -19864.349,E2 -19864.349} C_VEL
LIN {X 0,Y 236.046,Z 441.108,A -85,B 0,C 180,E1 -19866.764,E2 -19866.764} C_VEL
LIN {X 0,Y 233.267,Z 448.468,A -85,B 0,C 180,E1 -19869.248,E2 -19869.248} C_VEL
LIN {X 0,Y 230.459,Z 455.386,A -85,B 0,C 180,E1 -19872.243,E2 -19872.243} C_VEL
LIN {X 0,Y 228.534,Z 459.953,A -85,B 0,C 180,E1 -19874.845,E2 -19874.845} C_VEL
LIN {X 0,Y 227.16,Z 463.459,A -85,B 0,C 180,E1 -19877.49,E2 -19877.49} C_VEL
LIN {X 0,Y 226.551,Z 465.236,A -85,B 0,C 180,E1 -19879.271,E2 -19879.271} C_VEL
LIN {X 0,Y 225.771,Z 467.593,A -85,B 0,C 180,E1 -19882.845,E2 -19882.845} C_VEL
LIN {X 0,Y 225.696,Z 468.281,A -85,B 0,C 180,E1 -19885.181,E2 -19885.181} C_VEL
LIN {X 0,Y 225.83,Z 468.169,A -85,B 0,C 180,E1 -19888.214,E2 -19888.214} C_VEL
LIN {X 0,Y 225.881,Z 467.56,A -85,B 0,C 180,E1 -19889.997,E2 -19889.997} C_VEL
LIN {X 0,Y 225.866,Z 466.55,A -85,B 0,C 180,E1 -19891.78,E2 -19891.78} C_VEL
LIN {X 0,Y 225.796,Z 463.46,A -85,B 0,C 180,E1 -19895.112,E2 -19895.112} C_VEL
LIN {X 0,Y 225.969,Z 459.431,A -85,B 0,C 180,E1 -19898.042,E2 -19898.042} C_VEL
LIN {X 0,Y 226.408,Z 454.541,A -85,B 0,C 180,E1 -19900.73,E2 -19900.73} C_VEL
LIN {X 0,Y 227.236,Z 448.355,A -85,B 0,C 180,E1 -19903.408,E2 -19903.408} C_VEL
LIN {X 0,Y 228.489,Z 440.643,A -85,B 0,C 180,E1 -19906.066,E2 -19906.066} C_VEL
LIN {X 0,Y 229.789,Z 433.197,A -85,B 0,C 180,E1 -19908.14,E2 -19908.14} C_VEL
LIN {X 0,Y 231.654,Z 423.055,A -85,B 0,C 180,E1 -19910.414,E2 -19910.414} C_VEL
LIN {X 0,Y 233.376,Z 412.281,A -85,B 0,C 180,E1 -19912.34,E2 -19912.34} C_VEL
LIN {X 0,Y 234.992,Z 401.883,A -85,B 0,C 180,E1 -19913.807,E2 -19913.807} C_VEL
LIN {X 0,Y 236.451,Z 391.657,A -85,B 0,C 180,E1 -19914.936,E2 -19914.936} C_VEL
LIN {X 0,Y 237.897,Z 378.686,A -85,B 0,C 180,E1 -19916.003,E2 -19916.003} C_VEL
LIN {X 0,Y 238.942,Z 365.11,A -85,B 0,C 180,E1 -19916.746,E2 -19916.746} C_VEL
LIN {X 0,Y 240.743,Z 309.992,A -85,B 0,C 180,E1 -19918.4,E2 -19918.4} C_VEL
LIN {X 0,Y 236.059,Z 269.263,A -85,B 0,C 180,E1 -19920.221,E2 -19920.221} C_VEL
LIN {X 0,Y 230.982,Z 255.249,A -85,B 0,C 180,E1 -19921.293,E2 -19921.293} C_VEL
LIN {X 0,Y 228.56,Z 243.919,A -85,B 0,C 180,E1 -19925.741,E2 -19925.741} C_VEL
LIN {X 0,Y 227.918,Z 241.099,A -85,B 0,C 180,E1 -19926.936,E2 -19926.936} C_VEL
LIN {X 0,Y 227.811,Z 241.109,A -85,B 0,C 180,E1 -19930.371,E2 -19930.371} C_VEL
LIN {X 0,Y 227.835,Z 241.103,A -85,B 0,C 180,E1 -19935.183,E2 -19935.183} C_VEL
LIN {X 0,Y 227.887,Z 241.098,A -85,B 0,C 180,E1 -19937.734,E2 -19937.734} C_VEL
LIN {X 0,Y 227.847,Z 241.104,A -85,B 0,C 180,E1 -19941.909,E2 -19941.909} C_VEL
LIN {X 0,Y 227.856,Z 241.099,A -85,B 0,C 180,E1 -19946.373,E2 -19946.373} C_VEL
LIN {X 0,Y 227.893,Z 241.094,A -85,B 0,C 180,E1 -19950.433,E2 -19950.433} C_VEL
LIN {X 0,Y 227.902,Z 241.094,A -85,B 0,C 180,E1 -19954.422,E2 -19954.422} C_VEL
LIN {X 0,Y 227.976,Z 241.086,A -85,B 0,C 180,E1 -19958.288,E2 -19958.288} C_VEL
LIN {X 0,Y 228.002,Z 241.079,A -85,B 0,C 180,E1 -19962.826,E2 -19962.826} C_VEL
LIN {X 0,Y 228.027,Z 241.074,A -85,B 0,C 180,E1 -19967.54,E2 -19967.54} C_VEL
LIN {X 0,Y 228.272,Z 241.05,A -85,B 0,C 180,E1 -19971.144,E2 -19971.144} C_VEL
LIN {X 0,Y 228.319,Z 241.045,A -85,B 0,C 180,E1 -19972.927,E2 -19972.927} C_VEL
LIN {X 0,Y 228.516,Z 240.993,A -85,B 0,C 180,E1 -19978.237,E2 -19978.237} C_VEL
LIN {X 0,Y 228.514,Z 240.999,A -85,B 0,C 180,E1 -19981.762,E2 -19981.762} C_VEL
LIN {X 0,Y 228.282,Z 241.05,A -85,B 0,C 180,E1 -19987.073,E2 -19987.073} C_VEL
LIN {X 0,Y 228.107,Z 241.064,A -85,B 0,C 180,E1 -19990.652,E2 -19990.652} C_VEL
LIN {X 0,Y 227.997,Z 241.082,A -85,B 0,C 180,E1 -19994.276,E2 -19994.276} C_VEL
LIN {X 0,Y 227.896,Z 241.092,A -85,B 0,C 180,E1 -19997.961,E2 -19997.961} C_VEL
LIN {X 0,Y 227.866,Z 241.099,A -85,B 0,C 180,E1 -20002.31,E2 -20002.31} C_VEL
LIN {X 0,Y 227.903,Z 241.087,A -85,B 0,C 180,E1 -20006.6,E2 -20006.6} C_VEL
LIN {X 0,Y 227.848,Z 241.072,A -85,B 0,C 180,E1 -20010.285,E2 -20010.285} C_VEL
LIN {X 0,Y 227.85,Z 241.09,A -85,B 0,C 180,E1 -20013.724,E2 -20013.724} C_VEL
LIN {X 0,Y 227.819,Z 241.106,A -85,B 0,C 180,E1 -20018.095,E2 -20018.095} C_VEL
LIN {X 0,Y 227.78,Z 241.089,A -85,B 0,C 180,E1 -20022.749,E2 -20022.749} C_VEL
LIN {X 0,Y 227.783,Z 241.109,A -85,B 0,C 180,E1 -20027.26,E2 -20027.26} C_VEL
LIN {X 0,Y 227.826,Z 241.093,A -85,B 0,C 180,E1 -20031.913,E2 -20031.913} C_VEL
LIN {X 0,Y 227.864,Z 241.102,A -85,B 0,C 180,E1 -20036.382,E2 -20036.382} C_VEL
LIN {X 0,Y 227.891,Z 241.091,A -85,B 0,C 180,E1 -20040.44,E2 -20040.44} C_VEL
LIN {X 0,Y 227.914,Z 241.096,A -85,B 0,C 180,E1 -20044.43,E2 -20044.43} C_VEL
LIN {X 0,Y 227.93,Z 241.094,A -85,B 0,C 180,E1 -20048.289,E2 -20048.289} C_VEL
LIN {X 0,Y 228.012,Z 241.089,A -85,B 0,C 180,E1 -20053.61,E2 -20053.61} C_VEL
LIN {X 0,Y 229.119,Z 244.097,A -85,B 0,C 180,E1 -20053.853,E2 -20053.853} C_VEL
LIN {X 0,Y 237.411,Z 261.966,A -85,B 0,C 180,E1 -20055.42,E2 -20055.42} C_VEL
LIN {X 0,Y 241.699,Z 274.086,A -85,B 0,C 180,E1 -20056.276,E2 -20056.276} C_VEL
LIN {X 0,Y 239.748,Z 333.65,A -85,B 0,C 180,E1 -20058,E2 -20058} C_VEL
LIN {X 0,Y 239.048,Z 348.916,A -85,B 0,C 180,E1 -20058.558,E2 -20058.558} C_VEL
LIN {X 0,Y 238.186,Z 361.615,A -85,B 0,C 180,E1 -20059.377,E2 -20059.377} C_VEL
LIN {X 0,Y 237.048,Z 373.011,A -85,B 0,C 180,E1 -20060.404,E2 -20060.404} C_VEL
LIN {X 0,Y 235.501,Z 385.171,A -85,B 0,C 180,E1 -20061.854,E2 -20061.854} C_VEL
LIN {X 0,Y 233.796,Z 396.623,A -85,B 0,C 180,E1 -20063.646,E2 -20063.646} C_VEL
LIN {X 0,Y 232.05,Z 406.819,A -85,B 0,C 180,E1 -20065.661,E2 -20065.661} C_VEL
LIN {X 0,Y 230.454,Z 415.612,A -85,B 0,C 180,E1 -20067.819,E2 -20067.819} C_VEL
LIN {X 0,Y 228.885,Z 424.151,A -85,B 0,C 180,E1 -20070.443,E2 -20070.443} C_VEL
LIN {X 0,Y 227.682,Z 431,A -85,B 0,C 180,E1 -20073.099,E2 -20073.099} C_VEL
LIN {X 0,Y 226.746,Z 437.102,A -85,B 0,C 180,E1 -20076.126,E2 -20076.126} C_VEL
LIN {X 0,Y 226.094,Z 441.403,A -85,B 0,C 180,E1 -20078.944,E2 -20078.944} C_VEL
LIN {X 0,Y 225.78,Z 443.53,A -85,B 0,C 180,E1 -20080.766,E2 -20080.766} C_VEL
LIN {X 0,Y 225.619,Z 445.221,A -85,B 0,C 180,E1 -20082.596,E2 -20082.596} C_VEL
LIN {X 0,Y 225.571,Z 446.798,A -85,B 0,C 180,E1 -20085.019,E2 -20085.019} C_VEL
LIN {X 0,Y 225.758,Z 447.744,A -85,B 0,C 180,E1 -20088.14,E2 -20088.14} C_VEL
LIN {X 0,Y 226.433,Z 447.468,A -85,B 0,C 180,E1 -20091.389,E2 -20091.389} C_VEL
LIN {X 0,Y 227.135,Z 446.459,A -85,B 0,C 180,E1 -20093.72,E2 -20093.72} C_VEL
LIN {X 0,Y 228.621,Z 443.904,A -85,B 0,C 180,E1 -20096.941,E2 -20096.941} C_VEL
LIN {X 0,Y 230.66,Z 439.861,A -85,B 0,C 180,E1 -20100.182,E2 -20100.182} C_VEL
LIN {X 0,Y 232.9,Z 435.082,A -85,B 0,C 180,E1 -20102.9,E2 -20102.9} C_VEL
LIN {X 0,Y 235.577,Z 428.929,A -85,B 0,C 180,E1 -20105.573,E2 -20105.573} C_VEL
LIN {X 0,Y 238.681,Z 421.167,A -85,B 0,C 180,E1 -20108.195,E2 -20108.195} C_VEL
LIN {X 0,Y 241.526,Z 413.455,A -85,B 0,C 180,E1 -20110.251,E2 -20110.251} C_VEL
LIN {X 0,Y 244.507,Z 404.319,A -85,B 0,C 180,E1 -20112.211,E2 -20112.211} C_VEL
LIN {X 0,Y 247.723,Z 393.422,A -85,B 0,C 180,E1 -20114.032,E2 -20114.032} C_VEL
LIN {X 0,Y 250.258,Z 383.041,A -85,B 0,C 180,E1 -20115.407,E2 -20115.407} C_VEL
LIN {X 0,Y 252.524,Z 371.185,A -85,B 0,C 180,E1 -20116.641,E2 -20116.641} C_VEL
LIN {X 0,Y 254.484,Z 357.88,A -85,B 0,C 180,E1 -20117.623,E2 -20117.623} C_VEL
LIN {X 0,Y 255.665,Z 345.688,A -85,B 0,C 180,E1 -20118.237,E2 -20118.237} C_VEL
LIN {X 0,Y 258.143,Z 298.798,A -85,B 0,C 180,E1 -20119.54,E2 -20119.54} C_VEL
LIN {X 0,Y 258.454,Z 291.596,A -85,B 0,C 180,E1 -20119.744,E2 -20119.744} C_VEL
LIN {X 0,Y 252.248,Z 278.641,A -85,B 0,C 180,E1 -20121.461,E2 -20121.461} C_VEL
LIN {X 0,Y 247.433,Z 270.096,A -85,B 0,C 180,E1 -20122.832,E2 -20122.832} C_VEL
LIN {X 0,Y 239.735,Z 258.443,A -85,B 0,C 180,E1 -20125.135,E2 -20125.135} C_VEL
LIN {X 0,Y 236.596,Z 254.041,A -85,B 0,C 180,E1 -20126.138,E2 -20126.138} C_VEL
LIN {X 0,Y 234.135,Z 250.559,A -85,B 0,C 180,E1 -20126.958,E2 -20126.958} C_VEL
LIN {X 0,Y 231.911,Z 247.634,A -85,B 0,C 180,E1 -20127.716,E2 -20127.716} C_VEL
LIN {X 0,Y 231.187,Z 246.257,A -85,B 0,C 180,E1 -20127.989,E2 -20127.989} C_VEL
LIN {X 0,Y 228.952,Z 244.08,A -85,B 0,C 180,E1 -20128.751,E2 -20128.751} C_VEL
LIN {X 0,Y 227.891,Z 241.321,A -85,B 0,C 180,E1 -20129.207,E2 -20129.207} C_VEL
LIN {X 0,Y 227.885,Z 241.095,A -85,B 0,C 180,E1 -20129.542,E2 -20129.542} C_VEL
LIN {X 0,Y 227.92,Z 241.082,A -85,B 0,C 180,E1 -20134.425,E2 -20134.425} C_VEL
LIN {X 0,Y 227.953,Z 241.078,A -85,B 0,C 180,E1 -20138.287,E2 -20138.287} C_VEL
LIN {X 0,Y 228.025,Z 241.068,A -85,B 0,C 180,E1 -20142.828,E2 -20142.828} C_VEL
LIN {X 0,Y 228.049,Z 241.066,A -85,B 0,C 180,E1 -20147.542,E2 -20147.542} C_VEL
LIN {X 0,Y 228.241,Z 241.042,A -85,B 0,C 180,E1 -20151.144,E2 -20151.144} C_VEL
LIN {X 0,Y 228.306,Z 241.035,A -85,B 0,C 180,E1 -20152.928,E2 -20152.928} C_VEL
LIN {X 0,Y 228.537,Z 241.011,A -85,B 0,C 180,E1 -20158.238,E2 -20158.238} C_VEL
LIN {X 0,Y 228.536,Z 240.999,A -85,B 0,C 180,E1 -20161.763,E2 -20161.763} C_VEL
LIN {X 0,Y 228.288,Z 241.035,A -85,B 0,C 180,E1 -20167.074,E2 -20167.074} C_VEL
LIN {X 0,Y 228.118,Z 241.05,A -85,B 0,C 180,E1 -20170.653,E2 -20170.653} C_VEL
LIN {X 0,Y 228.008,Z 241.074,A -85,B 0,C 180,E1 -20176.106,E2 -20176.106} C_VEL
LIN {X 0,Y 227.914,Z 241.094,A -85,B 0,C 180,E1 -20181.718,E2 -20181.718} C_VEL
LIN {X 0,Y 227.872,Z 241.089,A -85,B 0,C 180,E1 -20183.502,E2 -20183.502} C_VEL
LIN {X 0,Y 227.239,Z 241.178,A -85,B 0,C 180,E1 -20184.978,E2 -20184.978} C_VEL
LIN {X 0,Y 224.399,Z 241.523,A -85,B 0,C 180,E1 -20187.386,E2 -20187.386} C_VEL
LIN {X 0,Y 221.95,Z 241.839,A -85,B 0,C 180,E1 -20189.35,E2 -20189.35} C_VEL
LIN {X 0,Y 220.878,Z 241.963,A -85,B 0,C 180,E1 -20190.875,E2 -20190.875} C_VEL
LIN {X 0,Y 220.781,Z 241.974,A -85,B 0,C 180,E1 -20191.393,E2 -20191.393} C_VEL
LIN {X 0,Y 220.785,Z 241.976,A -85,B 0,C 180,E1 -20194.959,E2 -20194.959} C_VEL
LIN {X 0,Y 220.82,Z 242.086,A -85,B 0,C 180,E1 -20197.926,E2 -20197.926} C_VEL
LIN {X 0,Y 222.867,Z 248.582,A -85,B 0,C 180,E1 -20202.304,E2 -20202.304} C_VEL
LIN {X 0,Y 224.068,Z 252.403,A -85,B 0,C 180,E1 -20204.573,E2 -20204.573} C_VEL
LIN {X 0,Y 227.151,Z 257.292,A -85,B 0,C 180,E1 -20205.771,E2 -20205.771} C_VEL
LIN {X 0,Y 232.055,Z 265.209,A -85,B 0,C 180,E1 -20207.561,E2 -20207.561} C_VEL
LIN {X 0,Y 237.484,Z 274.54,A -85,B 0,C 180,E1 -20209.414,E2 -20209.414} C_VEL
LIN {X 0,Y 243.649,Z 286.622,A -85,B 0,C 180,E1 -20211.4,E2 -20211.4} C_VEL
LIN {X 0,Y 248.921,Z 298.427,A -85,B 0,C 180,E1 -20213.024,E2 -20213.024} C_VEL
LIN {X 0,Y 249.757,Z 301.043,A -85,B 0,C 180,E1 -20213.3,E2 -20213.3} C_VEL
LIN {X 0,Y 251.926,Z 316.831,A -85,B 0,C 180,E1 -20214.34,E2 -20214.34} C_VEL
LIN {X 0,Y 249.462,Z 363.391,A -85,B 0,C 180,E1 -20215.663,E2 -20215.663} C_VEL
LIN {X 0,Y 247.838,Z 376.879,A -85,B 0,C 180,E1 -20216.307,E2 -20216.307} C_VEL
LIN {X 0,Y 245.687,Z 389.307,A -85,B 0,C 180,E1 -20217.199,E2 -20217.199} C_VEL
LIN {X 0,Y 242.952,Z 401.22,A -85,B 0,C 180,E1 -20218.378,E2 -20218.378} C_VEL
LIN {X 0,Y 239.751,Z 412.642,A -85,B 0,C 180,E1 -20219.867,E2 -20219.867} C_VEL
LIN {X 0,Y 236.439,Z 422.958,A -85,B 0,C 180,E1 -20221.602,E2 -20221.602} C_VEL
LIN {X 0,Y 233.12,Z 432.268,A -85,B 0,C 180,E1 -20223.597,E2 -20223.597} C_VEL
LIN {X 0,Y 229.542,Z 441.299,A -85,B 0,C 180,E1 -20226.065,E2 -20226.065} C_VEL
LIN {X 0,Y 226.439,Z 449.038,A -85,B 0,C 180,E1 -20228.793,E2 -20228.793} C_VEL
LIN {X 0,Y 223.675,Z 455.366,A -85,B 0,C 180,E1 -20231.686,E2 -20231.686} C_VEL
LIN {X 0,Y 221.68,Z 459.863,A -85,B 0,C 180,E1 -20234.365,E2 -20234.365} C_VEL
LIN {X 0,Y 220.182,Z 463.309,A -85,B 0,C 180,E1 -20237.087,E2 -20237.087} C_VEL
LIN {X 0,Y 219.043,Z 466.385,A -85,B 0,C 180,E1 -20240.766,E2 -20240.766} C_VEL
LIN {X 0,Y 218.591,Z 467.9,A -85,B 0,C 180,E1 -20244.462,E2 -20244.462} C_VEL
LIN {X 0,Y 218.757,Z 467.796,A -85,B 0,C 180,E1 -20248.156,E2 -20248.156} C_VEL
LIN {X 0,Y 218.812,Z 467.158,A -85,B 0,C 180,E1 -20249.997,E2 -20249.997} C_VEL
LIN {X 0,Y 218.773,Z 466.108,A -85,B 0,C 180,E1 -20251.838,E2 -20251.838} C_VEL
LIN {X 0,Y 218.717,Z 463.201,A -85,B 0,C 180,E1 -20255.044,E2 -20255.044} C_VEL
LIN {X 0,Y 218.898,Z 458.829,A -85,B 0,C 180,E1 -20258.303,E2 -20258.303} C_VEL
LIN {X 0,Y 219.375,Z 453.863,A -85,B 0,C 180,E1 -20261.078,E2 -20261.078} C_VEL
LIN {X 0,Y 220.276,Z 447.593,A -85,B 0,C 180,E1 -20263.84,E2 -20263.84} C_VEL
LIN {X 0,Y 221.626,Z 439.751,A -85,B 0,C 180,E1 -20266.578,E2 -20266.578} C_VEL
LIN {X 0,Y 222.772,Z 433.446,A -85,B 0,C 180,E1 -20268.385,E2 -20268.385} C_VEL
LIN {X 0,Y 224.573,Z 424.064,A -85,B 0,C 180,E1 -20270.609,E2 -20270.609} C_VEL
LIN {X 0,Y 226.268,Z 413.555,A -85,B 0,C 180,E1 -20272.599,E2 -20272.599} C_VEL
LIN {X 0,Y 228.211,Z 401.926,A -85,B 0,C 180,E1 -20274.318,E2 -20274.318} C_VEL
LIN {X 0,Y 229.711,Z 391.794,A -85,B 0,C 180,E1 -20275.477,E2 -20275.477} C_VEL
LIN {X 0,Y 231.201,Z 379.066,A -85,B 0,C 180,E1 -20276.572,E2 -20276.572} C_VEL
LIN {X 0,Y 232.295,Z 365.499,A -85,B 0,C 180,E1 -20277.349,E2 -20277.349} C_VEL
LIN {X 0,Y 233.448,Z 335.813,A -85,B 0,C 180,E1 -20278.289,E2 -20278.289} C_VEL
LIN {X 0,Y 234.147,Z 310.163,A -85,B 0,C 180,E1 -20279.068,E2 -20279.068} C_VEL
LIN {X 0,Y 229.76,Z 271.333,A -85,B 0,C 180,E1 -20280.865,E2 -20280.865} C_VEL
LIN {X 0,Y 223.64,Z 254.81,A -85,B 0,C 180,E1 -20282.232,E2 -20282.232} C_VEL
LIN {X 0,Y 221.404,Z 244.325,A -85,B 0,C 180,E1 -20286.517,E2 -20286.517} C_VEL
LIN {X 0,Y 220.847,Z 241.98,A -85,B 0,C 180,E1 -20287.531,E2 -20287.531} C_VEL
LIN {X 0,Y 220.755,Z 241.988,A -85,B 0,C 180,E1 -20291.947,E2 -20291.947} C_VEL
LIN {X 0,Y 220.845,Z 241.975,A -85,B 0,C 180,E1 -20297.038,E2 -20297.038} C_VEL
LIN {X 0,Y 220.835,Z 241.974,A -85,B 0,C 180,E1 -20300.469,E2 -20300.469} C_VEL
LIN {X 0,Y 220.78,Z 241.982,A -85,B 0,C 180,E1 -20305.041,E2 -20305.041} C_VEL
LIN {X 0,Y 220.844,Z 241.976,A -85,B 0,C 180,E1 -20309.391,E2 -20309.391} C_VEL
LIN {X 0,Y 220.869,Z 241.974,A -85,B 0,C 180,E1 -20313.545,E2 -20313.545} C_VEL
LIN {X 0,Y 220.907,Z 241.968,A -85,B 0,C 180,E1 -20317.556,E2 -20317.556} C_VEL
LIN {X 0,Y 220.952,Z 241.956,A -85,B 0,C 180,E1 -20322.571,E2 -20322.571} C_VEL
LIN {X 0,Y 220.966,Z 241.957,A -85,B 0,C 180,E1 -20327.135,E2 -20327.135} C_VEL
LIN {X 0,Y 221.203,Z 241.929,A -85,B 0,C 180,E1 -20330.859,E2 -20330.859} C_VEL
LIN {X 0,Y 221.255,Z 241.924,A -85,B 0,C 180,E1 -20332.7,E2 -20332.7} C_VEL
LIN {X 0,Y 221.474,Z 241.868,A -85,B 0,C 180,E1 -20338.181,E2 -20338.181} C_VEL
LIN {X 0,Y 221.448,Z 241.877,A -85,B 0,C 180,E1 -20341.818,E2 -20341.818} C_VEL
LIN {X 0,Y 221.216,Z 241.929,A -85,B 0,C 180,E1 -20347.3,E2 -20347.3} C_VEL
LIN {X 0,Y 221.028,Z 241.944,A -85,B 0,C 180,E1 -20350.998,E2 -20350.998} C_VEL
LIN {X 0,Y 220.943,Z 241.964,A -85,B 0,C 180,E1 -20356.635,E2 -20356.635} C_VEL
LIN {X 0,Y 220.818,Z 241.971,A -85,B 0,C 180,E1 -20360.493,E2 -20360.493} C_VEL
LIN {X 0,Y 220.823,Z 241.979,A -85,B 0,C 180,E1 -20364.44,E2 -20364.44} C_VEL
LIN {X 0,Y 220.782,Z 241.96,A -85,B 0,C 180,E1 -20368.521,E2 -20368.521} C_VEL
LIN {X 0,Y 220.785,Z 241.961,A -85,B 0,C 180,E1 -20372.761,E2 -20372.761} C_VEL
LIN {X 0,Y 220.785,Z 241.981,A -85,B 0,C 180,E1 -20377.282,E2 -20377.282} C_VEL
LIN {X 0,Y 220.739,Z 241.968,A -85,B 0,C 180,E1 -20381.959,E2 -20381.959} C_VEL
LIN {X 0,Y 220.746,Z 241.979,A -85,B 0,C 180,E1 -20385.548,E2 -20385.548} C_VEL
LIN {X 0,Y 220.767,Z 241.978,A -85,B 0,C 180,E1 -20390.463,E2 -20390.463} C_VEL
LIN {X 0,Y 220.808,Z 241.966,A -85,B 0,C 180,E1 -20392.798,E2 -20392.798} C_VEL
LIN {X 0,Y 220.802,Z 241.979,A -85,B 0,C 180,E1 -20397.249,E2 -20397.249} C_VEL
LIN {X 0,Y 220.814,Z 241.976,A -85,B 0,C 180,E1 -20401.49,E2 -20401.49} C_VEL
LIN {X 0,Y 220.851,Z 241.976,A -85,B 0,C 180,E1 -20405.569,E2 -20405.569} C_VEL
LIN {X 0,Y 220.861,Z 241.975,A -85,B 0,C 180,E1 -20409.516,E2 -20409.516} C_VEL
LIN {X 0,Y 220.941,Z 241.969,A -85,B 0,C 180,E1 -20412.734,E2 -20412.734} C_VEL
LIN {X 0,Y 221.957,Z 244.837,A -85,B 0,C 180,E1 -20412.977,E2 -20412.977} C_VEL
LIN {X 0,Y 229.65,Z 260.88,A -85,B 0,C 180,E1 -20414.495,E2 -20414.495} C_VEL
LIN {X 0,Y 233.827,Z 271.415,A -85,B 0,C 180,E1 -20415.337,E2 -20415.337} C_VEL
LIN {X 0,Y 235.289,Z 276.081,A -85,B 0,C 180,E1 -20415.655,E2 -20415.655} C_VEL
LIN {X 0,Y 232.75,Z 343.965,A -85,B 0,C 180,E1 -20417.686,E2 -20417.686} C_VEL
LIN {X 0,Y 231.923,Z 357.253,A -85,B 0,C 180,E1 -20418.423,E2 -20418.423} C_VEL
LIN {X 0,Y 230.697,Z 369.98,A -85,B 0,C 180,E1 -20419.472,E2 -20419.472} C_VEL
LIN {X 0,Y 229.301,Z 381.31,A -85,B 0,C 180,E1 -20420.744,E2 -20420.744} C_VEL
LIN {X 0,Y 227.671,Z 392.955,A -85,B 0,C 180,E1 -20422.465,E2 -20422.465} C_VEL
LIN {X 0,Y 226.028,Z 402.648,A -85,B 0,C 180,E1 -20424.257,E2 -20424.257} C_VEL
LIN {X 0,Y 224.257,Z 412.072,A -85,B 0,C 180,E1 -20426.41,E2 -20426.41} C_VEL
LIN {X 0,Y 222.712,Z 420,A -85,B 0,C 180,E1 -20428.647,E2 -20428.647} C_VEL
LIN {X 0,Y 221.272,Z 427.722,A -85,B 0,C 180,E1 -20431.368,E2 -20431.368} C_VEL
LIN {X 0,Y 220.356,Z 433.008,A -85,B 0,C 180,E1 -20433.66,E2 -20433.66} C_VEL
LIN {X 0,Y 219.455,Z 438.849,A -85,B 0,C 180,E1 -20436.899,E2 -20436.899} C_VEL
LIN {X 0,Y 218.776,Z 443.21,A -85,B 0,C 180,E1 -20440.179,E2 -20440.179} C_VEL
LIN {X 0,Y 218.515,Z 445.805,A -85,B 0,C 180,E1 -20443.013,E2 -20443.013} C_VEL
LIN {X 0,Y 218.492,Z 447.135,A -85,B 0,C 180,E1 -20445.211,E2 -20445.211} C_VEL
LIN {X 0,Y 218.744,Z 448.11,A -85,B 0,C 180,E1 -20448.742,E2 -20448.742} C_VEL
LIN {X 0,Y 219.414,Z 447.808,A -85,B 0,C 180,E1 -20451.739,E2 -20451.739} C_VEL
LIN {X 0,Y 220.329,Z 446.6,A -85,B 0,C 180,E1 -20454.5,E2 -20454.5} C_VEL
LIN {X 0,Y 221.77,Z 444.267,A -85,B 0,C 180,E1 -20457.461,E2 -20457.461} C_VEL
LIN {X 0,Y 223.505,Z 441.05,A -85,B 0,C 180,E1 -20460.207,E2 -20460.207} C_VEL
LIN {X 0,Y 225.896,Z 436.333,A -85,B 0,C 180,E1 -20463.136,E2 -20463.136} C_VEL
LIN {X 0,Y 228.482,Z 430.769,A -85,B 0,C 180,E1 -20465.763,E2 -20465.763} C_VEL
LIN {X 0,Y 231.57,Z 423.657,A -85,B 0,C 180,E1 -20468.363,E2 -20468.363} C_VEL
LIN {X 0,Y 234.657,Z 415.747,A -85,B 0,C 180,E1 -20470.648,E2 -20470.648} C_VEL
LIN {X 0,Y 237.981,Z 406.413,A -85,B 0,C 180,E1 -20472.783,E2 -20472.783} C_VEL
LIN {X 0,Y 241.288,Z 396.023,A -85,B 0,C 180,E1 -20474.642,E2 -20474.642} C_VEL
LIN {X 0,Y 244.136,Z 385.163,A -85,B 0,C 180,E1 -20476.165,E2 -20476.165} C_VEL
LIN {X 0,Y 246.619,Z 373.038,A -85,B 0,C 180,E1 -20477.495,E2 -20477.495} C_VEL
LIN {X 0,Y 248.684,Z 360.395,A -85,B 0,C 180,E1 -20478.494,E2 -20478.494} C_VEL
LIN {X 0,Y 250.068,Z 347.269,A -85,B 0,C 180,E1 -20479.204,E2 -20479.204} C_VEL
LIN {X 0,Y 251.408,Z 324.845,A -85,B 0,C 180,E1 -20479.876,E2 -20479.876} C_VEL
LIN {X 0,Y 253.021,Z 293.933,A -85,B 0,C 180,E1 -20480.721,E2 -20480.721} C_VEL
LIN {X 0,Y 246.406,Z 280.338,A -85,B 0,C 180,E1 -20482.651,E2 -20482.651} C_VEL
LIN {X 0,Y 240.768,Z 270.958,A -85,B 0,C 180,E1 -20484.347,E2 -20484.347} C_VEL
LIN {X 0,Y 233.659,Z 260.254,A -85,B 0,C 180,E1 -20486.643,E2 -20486.643} C_VEL
LIN {X 0,Y 230.319,Z 255.713,A -85,B 0,C 180,E1 -20487.789,E2 -20487.789} C_VEL
LIN {X 0,Y 227.57,Z 251.842,A -85,B 0,C 180,E1 -20488.786,E2 -20488.786} C_VEL
LIN {X 0,Y 225.329,Z 249.147,A -85,B 0,C 180,E1 -20489.61,E2 -20489.61} C_VEL
LIN {X 0,Y 224.282,Z 247.213,A -85,B 0,C 180,E1 -20490.04,E2 -20490.04} C_VEL
LIN {X 0,Y 221.929,Z 244.986,A -85,B 0,C 180,E1 -20490.929,E2 -20490.929} C_VEL
LIN {X 0,Y 220.876,Z 242.38,A -85,B 0,C 180,E1 -20491.428,E2 -20491.428} C_VEL
LIN {X 0,Y 220.803,Z 241.968,A -85,B 0,C 180,E1 -20491.482,E2 -20491.482} C_VEL
LIN {X 0,Y 220.859,Z 241.96,A -85,B 0,C 180,E1 -20495.565,E2 -20495.565} C_VEL
LIN {X 0,Y 220.883,Z 241.958,A -85,B 0,C 180,E1 -20499.514,E2 -20499.514} C_VEL
LIN {X 0,Y 221.004,Z 241.943,A -85,B 0,C 180,E1 -20503.37,E2 -20503.37} C_VEL
LIN {X 0,Y 221.053,Z 241.947,A -85,B 0,C 180,E1 -20509.003,E2 -20509.003} C_VEL
LIN {X 0,Y 221.241,Z 241.913,A -85,B 0,C 180,E1 -20512.701,E2 -20512.701} C_VEL
LIN {X 0,Y 221.495,Z 241.887,A -85,B 0,C 180,E1 -20518.182,E2 -20518.182} C_VEL
LIN {X 0,Y 221.47,Z 241.879,A -85,B 0,C 180,E1 -20521.819,E2 -20521.819} C_VEL
LIN {X 0,Y 221.225,Z 241.916,A -85,B 0,C 180,E1 -20527.301,E2 -20527.301} C_VEL
LIN {X 0,Y 221.044,Z 241.933,A -85,B 0,C 180,E1 -20530.998,E2 -20530.998} C_VEL
LIN {X 0,Y 220.967,Z 241.956,A -85,B 0,C 180,E1 -20536.634,E2 -20536.634} C_VEL
LIN {X 0,Y 220.84,Z 241.97,A -85,B 0,C 180,E1 -20540.492,E2 -20540.492} C_VEL
LIN {X 0,Y 220.834,Z 241.97,A -85,B 0,C 180,E1 -20544.44,E2 -20544.44} C_VEL
LIN {X 0,Y 220.796,Z 241.977,A -85,B 0,C 180,E1 -20548.52,E2 -20548.52} C_VEL
LIN {X 0,Y 220.781,Z 241.974,A -85,B 0,C 180,E1 -20551.393,E2 -20551.393} C_VEL
LIN {X 0,Y 220.041,Z 242.078,A -85,B 0,C 180,E1 -20552.421,E2 -20552.421} C_VEL
LIN {X 0,Y 217.093,Z 242.436,A -85,B 0,C 180,E1 -20554.036,E2 -20554.036} C_VEL
LIN {X 0,Y 214.423,Z 243.25,A -85,B 0,C 180,E1 -20555.666,E2 -20555.666} C_VEL
LIN {X 0,Y 214.106,Z 244.239,A -85,B 0,C 180,E1 -20556.685,E2 -20556.685} C_VEL
LIN {X 0,Y 215.908,Z 249.63,A -85,B 0,C 180,E1 -20560.619,E2 -20560.619} C_VEL
LIN {X 0,Y 216.683,Z 251.905,A -85,B 0,C 180,E1 -20562.027,E2 -20562.027} C_VEL
LIN {X 0,Y 219.575,Z 256.468,A -85,B 0,C 180,E1 -20563.302,E2 -20563.302} C_VEL
LIN {X 0,Y 221.144,Z 258.724,A -85,B 0,C 180,E1 -20563.952,E2 -20563.952} C_VEL
LIN {X 0,Y 225.177,Z 265.102,A -85,B 0,C 180,E1 -20565.558,E2 -20565.558} C_VEL
LIN {X 0,Y 229.275,Z 271.941,A -85,B 0,C 180,E1 -20567.098,E2 -20567.098} C_VEL
LIN {X 0,Y 234.055,Z 280.48,A -85,B 0,C 180,E1 -20568.796,E2 -20568.796} C_VEL
LIN {X 0,Y 239.529,Z 291.508,A -85,B 0,C 180,E1 -20570.64,E2 -20570.64} C_VEL
LIN {X 0,Y 244.539,Z 303.039,A -85,B 0,C 180,E1 -20572.265,E2 -20572.265} C_VEL
LIN {X 0,Y 246.547,Z 317.947,A -85,B 0,C 180,E1 -20573.288,E2 -20573.288} C_VEL
LIN {X 0,Y 244.07,Z 363.015,A -85,B 0,C 180,E1 -20574.589,E2 -20574.589} C_VEL
LIN {X 0,Y 242.373,Z 376.692,A -85,B 0,C 180,E1 -20575.252,E2 -20575.252} C_VEL
LIN {X 0,Y 240.011,Z 389.611,A -85,B 0,C 180,E1 -20576.196,E2 -20576.196} C_VEL
LIN {X 0,Y 236.984,Z 402.144,A -85,B 0,C 180,E1 -20577.485,E2 -20577.485} C_VEL
LIN {X 0,Y 233.681,Z 413.337,A -85,B 0,C 180,E1 -20579,E2 -20579} C_VEL
LIN {X 0,Y 230.257,Z 423.454,A -85,B 0,C 180,E1 -20580.767,E2 -20580.767} C_VEL
LIN {X 0,Y 226.794,Z 432.586,A -85,B 0,C 180,E1 -20582.8,E2 -20582.8} C_VEL
LIN {X 0,Y 223.073,Z 441.51,A -85,B 0,C 180,E1 -20585.325,E2 -20585.325} C_VEL
LIN {X 0,Y 220.172,Z 448.281,A -85,B 0,C 180,E1 -20587.775,E2 -20587.775} C_VEL
LIN {X 0,Y 217.754,Z 453.624,A -85,B 0,C 180,E1 -20590.189,E2 -20590.189} C_VEL
LIN {X 0,Y 215.503,Z 458.419,A -85,B 0,C 180,E1 -20592.93,E2 -20592.93} C_VEL
LIN {X 0,Y 213.682,Z 462.126,A -85,B 0,C 180,E1 -20595.717,E2 -20595.717} C_VEL
LIN {X 0,Y 212.532,Z 464.853,A -85,B 0,C 180,E1 -20598.554,E2 -20598.554} C_VEL
LIN {X 0,Y 211.639,Z 467.085,A -85,B 0,C 180,E1 -20602.364,E2 -20602.364} C_VEL
LIN {X 0,Y 211.516,Z 467.716,A -85,B 0,C 180,E1 -20605.424,E2 -20605.424} C_VEL
LIN {X 0,Y 211.662,Z 467.422,A -85,B 0,C 180,E1 -20608.094,E2 -20608.094} C_VEL
LIN {X 0,Y 211.745,Z 466.755,A -85,B 0,C 180,E1 -20609.997,E2 -20609.997} C_VEL
LIN {X 0,Y 211.682,Z 465.646,A -85,B 0,C 180,E1 -20611.899,E2 -20611.899} C_VEL
LIN {X 0,Y 211.621,Z 463.002,A -85,B 0,C 180,E1 -20614.916,E2 -20614.916} C_VEL
LIN {X 0,Y 211.745,Z 459.665,A -85,B 0,C 180,E1 -20617.625,E2 -20617.625} C_VEL
LIN {X 0,Y 212.148,Z 455.02,A -85,B 0,C 180,E1 -20620.494,E2 -20620.494} C_VEL
LIN {X 0,Y 213.161,Z 447.967,A -85,B 0,C 180,E1 -20623.825,E2 -20623.825} C_VEL
LIN {X 0,Y 214.498,Z 440.314,A -85,B 0,C 180,E1 -20626.655,E2 -20626.655} C_VEL
LIN {X 0,Y 215.718,Z 434.145,A -85,B 0,C 180,E1 -20628.516,E2 -20628.516} C_VEL
LIN {X 0,Y 216.963,Z 427.405,A -85,B 0,C 180,E1 -20630.261,E2 -20630.261} C_VEL
LIN {X 0,Y 218.83,Z 417.252,A -85,B 0,C 180,E1 -20632.414,E2 -20632.414} C_VEL
LIN {X 0,Y 220.71,Z 406.656,A -85,B 0,C 180,E1 -20634.197,E2 -20634.197} C_VEL
LIN {X 0,Y 222.641,Z 394.959,A -85,B 0,C 180,E1 -20635.718,E2 -20635.718} C_VEL
LIN {X 0,Y 224.193,Z 382.76,A -85,B 0,C 180,E1 -20636.904,E2 -20636.904} C_VEL
LIN {X 0,Y 225.481,Z 369.499,A -85,B 0,C 180,E1 -20637.805,E2 -20637.805} C_VEL
LIN {X 0,Y 226.19,Z 356.658,A -85,B 0,C 180,E1 -20638.337,E2 -20638.337} C_VEL
LIN {X 0,Y 227.617,Z 310.531,A -85,B 0,C 180,E1 -20639.764,E2 -20639.764} C_VEL
LIN {X 0,Y 223.447,Z 273.37,A -85,B 0,C 180,E1 -20641.551,E2 -20641.551} C_VEL
LIN {X 0,Y 217.392,Z 257.388,A -85,B 0,C 180,E1 -20642.903,E2 -20642.903} C_VEL
LIN {X 0,Y 216.343,Z 254.483,A -85,B 0,C 180,E1 -20643.189,E2 -20643.189} C_VEL
LIN {X 0,Y 214.593,Z 246.276,A -85,B 0,C 180,E1 -20646.67,E2 -20646.67} C_VEL
LIN {X 0,Y 213.785,Z 242.86,A -85,B 0,C 180,E1 -20648.197,E2 -20648.197} C_VEL
LIN {X 0,Y 213.697,Z 242.866,A -85,B 0,C 180,E1 -20651.12,E2 -20651.12} C_VEL
LIN {X 0,Y 213.762,Z 242.858,A -85,B 0,C 180,E1 -20656.335,E2 -20656.335} C_VEL
LIN {X 0,Y 213.775,Z 242.856,A -85,B 0,C 180,E1 -20659.114,E2 -20659.114} C_VEL
LIN {X 0,Y 213.724,Z 242.86,A -85,B 0,C 180,E1 -20663.707,E2 -20663.707} C_VEL
LIN {X 0,Y 213.757,Z 242.856,A -85,B 0,C 180,E1 -20668.727,E2 -20668.727} C_VEL
LIN {X 0,Y 213.802,Z 242.85,A -85,B 0,C 180,E1 -20672.599,E2 -20672.599} C_VEL
LIN {X 0,Y 213.839,Z 242.844,A -85,B 0,C 180,E1 -20676.941,E2 -20676.941} C_VEL
LIN {X 0,Y 213.902,Z 242.834,A -85,B 0,C 180,E1 -20682.304,E2 -20682.304} C_VEL
LIN {X 0,Y 213.908,Z 242.838,A -85,B 0,C 180,E1 -20686.703,E2 -20686.703} C_VEL
LIN {X 0,Y 214.135,Z 242.808,A -85,B 0,C 180,E1 -20690.554,E2 -20690.554} C_VEL
LIN {X 0,Y 214.193,Z 242.802,A -85,B 0,C 180,E1 -20692.458,E2 -20692.458} C_VEL
LIN {X 0,Y 214.407,Z 242.746,A -85,B 0,C 180,E1 -20698.121,E2 -20698.121} C_VEL
LIN {X 0,Y 214.508,Z 242.725,A -85,B 0,C 180,E1 -20699.999,E2 -20699.999} C_VEL
LIN {X 0,Y 214.385,Z 242.756,A -85,B 0,C 180,E1 -20701.878,E2 -20701.878} C_VEL
LIN {X 0,Y 214.155,Z 242.807,A -85,B 0,C 180,E1 -20707.542,E2 -20707.542} C_VEL
LIN {X 0,Y 213.959,Z 242.823,A -85,B 0,C 180,E1 -20711.366,E2 -20711.366} C_VEL
LIN {X 0,Y 213.863,Z 242.845,A -85,B 0,C 180,E1 -20715.241,E2 -20715.241} C_VEL
LIN {X 0,Y 213.763,Z 242.847,A -85,B 0,C 180,E1 -20719.194,E2 -20719.194} C_VEL
LIN {X 0,Y 213.765,Z 242.856,A -85,B 0,C 180,E1 -20723.236,E2 -20723.236} C_VEL
LIN {X 0,Y 213.766,Z 242.843,A -85,B 0,C 180,E1 -20727.434,E2 -20727.434} C_VEL
LIN {X 0,Y 213.732,Z 242.831,A -85,B 0,C 180,E1 -20731.743,E2 -20731.743} C_VEL
LIN {X 0,Y 213.719,Z 242.861,A -85,B 0,C 180,E1 -20736.292,E2 -20736.292} C_VEL
LIN {X 0,Y 213.682,Z 242.852,A -85,B 0,C 180,E1 -20741.131,E2 -20741.131} C_VEL
LIN {X 0,Y 213.682,Z 242.844,A -85,B 0,C 180,E1 -20743.684,E2 -20743.684} C_VEL
LIN {X 0,Y 213.683,Z 242.863,A -85,B 0,C 180,E1 -20746.35,E2 -20746.35} C_VEL
LIN {X 0,Y 213.69,Z 242.865,A -85,B 0,C 180,E1 -20749.151,E2 -20749.151} C_VEL
LIN {X 0,Y 213.728,Z 242.851,A -85,B 0,C 180,E1 -20753.716,E2 -20753.716} C_VEL
LIN {X 0,Y 213.767,Z 242.848,A -85,B 0,C 180,E1 -20758.736,E2 -20758.736} C_VEL
LIN {X 0,Y 213.815,Z 242.851,A -85,B 0,C 180,E1 -20762.608,E2 -20762.608} C_VEL
LIN {X 0,Y 213.809,Z 242.851,A -85,B 0,C 180,E1 -20766.979,E2 -20766.979} C_VEL
LIN {X 0,Y 213.87,Z 242.85,A -85,B 0,C 180,E1 -20771.796,E2 -20771.796} C_VEL
LIN {X 0,Y 214.969,Z 245.875,A -85,B 0,C 180,E1 -20772.075,E2 -20772.075} C_VEL
LIN {X 0,Y 222.633,Z 261.461,A -85,B 0,C 180,E1 -20773.662,E2 -20773.662} C_VEL
LIN {X 0,Y 227.679,Z 273.874,A -85,B 0,C 180,E1 -20774.712,E2 -20774.712} C_VEL
LIN {X 0,Y 228.788,Z 277.939,A -85,B 0,C 180,E1 -20774.982,E2 -20774.982} C_VEL
LIN {X 0,Y 226.143,Z 345.21,A -85,B 0,C 180,E1 -20777.059,E2 -20777.059} C_VEL
LIN {X 0,Y 225.243,Z 358.632,A -85,B 0,C 180,E1 -20777.846,E2 -20777.846} C_VEL
LIN {X 0,Y 224.004,Z 371.061,A -85,B 0,C 180,E1 -20778.925,E2 -20778.925} C_VEL
LIN {X 0,Y 222.534,Z 382.186,A -85,B 0,C 180,E1 -20780.231,E2 -20780.231} C_VEL
LIN {X 0,Y 220.839,Z 393.729,A -85,B 0,C 180,E1 -20782.001,E2 -20782.001} C_VEL
LIN {X 0,Y 218.849,Z 404.862,A -85,B 0,C 180,E1 -20784.165,E2 -20784.165} C_VEL
LIN {X 0,Y 217.142,Z 413.554,A -85,B 0,C 180,E1 -20786.292,E2 -20786.292} C_VEL
LIN {X 0,Y 215.337,Z 422.624,A -85,B 0,C 180,E1 -20789.068,E2 -20789.068} C_VEL
LIN {X 0,Y 213.902,Z 429.938,A -85,B 0,C 180,E1 -20791.886,E2 -20791.886} C_VEL
LIN {X 0,Y 212.885,Z 435.776,A -85,B 0,C 180,E1 -20794.737,E2 -20794.737} C_VEL
LIN {X 0,Y 212.165,Z 440.374,A -85,B 0,C 180,E1 -20797.617,E2 -20797.617} C_VEL
LIN {X 0,Y 211.628,Z 443.886,A -85,B 0,C 180,E1 -20800.527,E2 -20800.527} C_VEL
LIN {X 0,Y 211.39,Z 446.379,A -85,B 0,C 180,E1 -20803.46,E2 -20803.46} C_VEL
LIN {X 0,Y 211.395,Z 447.477,A -85,B 0,C 180,E1 -20805.426,E2 -20805.426} C_VEL
LIN {X 0,Y 211.493,Z 448.177,A -85,B 0,C 180,E1 -20807.404,E2 -20807.404} C_VEL
LIN {X 0,Y 211.751,Z 448.476,A -85,B 0,C 180,E1 -20809.386,E2 -20809.386} C_VEL
LIN {X 0,Y 212.434,Z 448.143,A -85,B 0,C 180,E1 -20812.132,E2 -20812.132} C_VEL
LIN {X 0,Y 213.562,Z 446.743,A -85,B 0,C 180,E1 -20815.33,E2 -20815.33} C_VEL
LIN {X 0,Y 214.974,Z 444.615,A -85,B 0,C 180,E1 -20818.032,E2 -20818.032} C_VEL
LIN {X 0,Y 217.055,Z 440.957,A -85,B 0,C 180,E1 -20821.203,E2 -20821.203} C_VEL
LIN {X 0,Y 219.467,Z 436.45,A -85,B 0,C 180,E1 -20824.014,E2 -20824.014} C_VEL
LIN {X 0,Y 222.463,Z 430.36,A -85,B 0,C 180,E1 -20826.887,E2 -20826.887} C_VEL
LIN {X 0,Y 225.859,Z 422.773,A -85,B 0,C 180,E1 -20829.635,E2 -20829.635} C_VEL
LIN {X 0,Y 229.056,Z 414.959,A -85,B 0,C 180,E1 -20831.862,E2 -20831.862} C_VEL
LIN {X 0,Y 232.553,Z 405.378,A -85,B 0,C 180,E1 -20834.033,E2 -20834.033} C_VEL
LIN {X 0,Y 236.049,Z 394.574,A -85,B 0,C 180,E1 -20835.912,E2 -20835.912} C_VEL
LIN {X 0,Y 239.002,Z 383.408,A -85,B 0,C 180,E1 -20837.443,E2 -20837.443} C_VEL
LIN {X 0,Y 241.383,Z 371.872,A -85,B 0,C 180,E1 -20838.675,E2 -20838.675} C_VEL
LIN {X 0,Y 243.454,Z 358.893,A -85,B 0,C 180,E1 -20839.665,E2 -20839.665} C_VEL
LIN {X 0,Y 244.815,Z 346.148,A -85,B 0,C 180,E1 -20840.323,E2 -20840.323} C_VEL
LIN {X 0,Y 247.61,Z 296.336,A -85,B 0,C 180,E1 -20841.75,E2 -20841.75} C_VEL
LIN {X 0,Y 241.744,Z 284.184,A -85,B 0,C 180,E1 -20843.56,E2 -20843.56} C_VEL
LIN {X 0,Y 235.147,Z 273.242,A -85,B 0,C 180,E1 -20845.659,E2 -20845.659} C_VEL
LIN {X 0,Y 227.618,Z 262.03,A -85,B 0,C 180,E1 -20848.274,E2 -20848.274} C_VEL
LIN {X 0,Y 223.895,Z 257.137,A -85,B 0,C 180,E1 -20849.657,E2 -20849.657} C_VEL
LIN {X 0,Y 221.384,Z 253.538,A -85,B 0,C 180,E1 -20850.66,E2 -20850.66} C_VEL
LIN {X 0,Y 218.438,Z 250.011,A -85,B 0,C 180,E1 -20851.866,E2 -20851.866} C_VEL
LIN {X 0,Y 217.507,Z 248.243,A -85,B 0,C 180,E1 -20852.298,E2 -20852.298} C_VEL
LIN {X 0,Y 215.115,Z 246.105,A -85,B 0,C 180,E1 -20853.307,E2 -20853.307} C_VEL
LIN {X 0,Y 213.993,Z 243.721,A -85,B 0,C 180,E1 -20853.878,E2 -20853.878} C_VEL
LIN {X 0,Y 213.829,Z 242.839,A -85,B 0,C 180,E1 -20854.053,E2 -20854.053} C_VEL
LIN {X 0,Y 213.845,Z 242.845,A -85,B 0,C 180,E1 -20856.954,E2 -20856.954} C_VEL
LIN {X 0,Y 213.934,Z 242.823,A -85,B 0,C 180,E1 -20862.803,E2 -20862.803} C_VEL
LIN {X 0,Y 213.932,Z 242.826,A -85,B 0,C 180,E1 -20866.706,E2 -20866.706} C_VEL
LIN {X 0,Y 214.118,Z 242.806,A -85,B 0,C 180,E1 -20870.555,E2 -20870.555} C_VEL
LIN {X 0,Y 214.081,Z 242.815,A -85,B 0,C 180,E1 -20874.349,E2 -20874.349} C_VEL
LIN {X 0,Y 214.429,Z 242.765,A -85,B 0,C 180,E1 -20878.122,E2 -20878.122} C_VEL
LIN {X 0,Y 214.528,Z 242.748,A -85,B 0,C 180,E1 -20880.001,E2 -20880.001} C_VEL
LIN {X 0,Y 214.407,Z 242.759,A -85,B 0,C 180,E1 -20881.879,E2 -20881.879} C_VEL
LIN {X 0,Y 214.167,Z 242.798,A -85,B 0,C 180,E1 -20887.543,E2 -20887.543} C_VEL
LIN {X 0,Y 213.977,Z 242.815,A -85,B 0,C 180,E1 -20891.366,E2 -20891.366} C_VEL
LIN {X 0,Y 213.872,Z 242.828,A -85,B 0,C 180,E1 -20895.242,E2 -20895.242} C_VEL
LIN {X 0,Y 213.784,Z 242.841,A -85,B 0,C 180,E1 -20899.193,E2 -20899.193} C_VEL
LIN {X 0,Y 213.786,Z 242.843,A -85,B 0,C 180,E1 -20903.235,E2 -20903.235} C_VEL
LIN {X 0,Y 213.781,Z 242.845,A -85,B 0,C 180,E1 -20907.428,E2 -20907.428} C_VEL
LIN {X 0,Y 213.752,Z 242.851,A -85,B 0,C 180,E1 -20911.741,E2 -20911.741} C_VEL
LIN {X 0,Y 213.727,Z 242.867,A -85,B 0,C 180,E1 -20915.636,E2 -20915.636} C_VEL
LIN {X 0,Y 214.106,Z 244.239,A -85,B 0,C 180,E1 -20916.685,E2 -20916.685} C_VEL
LIN {X 0,Y 214.66,Z 246.623,A -85,B 0,C 180,E1 -20918.125,E2 -20918.125} C_VEL
LIN {X 0,Y 214.996,Z 249.848,A -85,B 0,C 180,E1 -20919.453,E2 -20919.453} C_VEL
LIN {X 0,Y 215.533,Z 255.064,A -85,B 0,C 180,E1 -20921.05,E2 -20921.05} C_VEL
LIN {X 0,Y 216.714,Z 260.938,A -85,B 0,C 180,E1 -20922.453,E2 -20922.453} C_VEL
LIN {X 0,Y 217.746,Z 263.991,A -85,B 0,C 180,E1 -20923.076,E2 -20923.076} C_VEL
LIN {X 0,Y 222.041,Z 271.008,A -85,B 0,C 180,E1 -20924.877,E2 -20924.877} C_VEL
LIN {X 0,Y 226.901,Z 279.236,A -85,B 0,C 180,E1 -20926.764,E2 -20926.764} C_VEL
LIN {X 0,Y 233.19,Z 291.355,A -85,B 0,C 180,E1 -20929.057,E2 -20929.057} C_VEL
LIN {X 0,Y 239.077,Z 304.657,A -85,B 0,C 180,E1 -20931.085,E2 -20931.085} C_VEL
LIN {X 0,Y 239.81,Z 307.367,A -85,B 0,C 180,E1 -20931.37,E2 -20931.37} C_VEL
LIN {X 0,Y 241.264,Z 319.398,A -85,B 0,C 180,E1 -20932.199,E2 -20932.199} C_VEL
LIN {X 0,Y 238.722,Z 363.233,A -85,B 0,C 180,E1 -20933.491,E2 -20933.491} C_VEL
LIN {X 0,Y 237.001,Z 376.529,A -85,B 0,C 180,E1 -20934.15,E2 -20934.15} C_VEL
LIN {X 0,Y 234.674,Z 388.866,A -85,B 0,C 180,E1 -20935.058,E2 -20935.058} C_VEL
LIN {X 0,Y 231.504,Z 401.498,A -85,B 0,C 180,E1 -20936.356,E2 -20936.356} C_VEL
LIN {X 0,Y 228.086,Z 412.747,A -85,B 0,C 180,E1 -20937.891,E2 -20937.891} C_VEL
LIN {X 0,Y 224.486,Z 422.923,A -85,B 0,C 180,E1 -20939.68,E2 -20939.68} C_VEL
LIN {X 0,Y 220.513,Z 432.905,A -85,B 0,C 180,E1 -20941.959,E2 -20941.959} C_VEL
LIN {X 0,Y 216.653,Z 441.72,A -85,B 0,C 180,E1 -20944.543,E2 -20944.543} C_VEL
LIN {X 0,Y 213.433,Z 448.794,A -85,B 0,C 180,E1 -20947.221,E2 -20947.221} C_VEL
LIN {X 0,Y 211.086,Z 453.656,A -85,B 0,C 180,E1 -20949.536,E2 -20949.536} C_VEL
LIN {X 0,Y 208.721,Z 458.374,A -85,B 0,C 180,E1 -20952.358,E2 -20952.358} C_VEL
LIN {X 0,Y 206.796,Z 462.009,A -85,B 0,C 180,E1 -20955.231,E2 -20955.231} C_VEL
LIN {X 0,Y 205.536,Z 464.666,A -85,B 0,C 180,E1 -20958.159,E2 -20958.159} C_VEL
LIN {X 0,Y 204.982,Z 465.944,A -85,B 0,C 180,E1 -20960.127,E2 -20960.127} C_VEL
LIN {X 0,Y 204.6,Z 466.816,A -85,B 0,C 180,E1 -20962.1,E2 -20962.1} C_VEL
LIN {X 0,Y 204.427,Z 467.351,A -85,B 0,C 180,E1 -20966.054,E2 -20966.054} C_VEL
LIN {X 0,Y 204.569,Z 467.048,A -85,B 0,C 180,E1 -20968.028,E2 -20968.028} C_VEL
LIN {X 0,Y 204.678,Z 466.346,A -85,B 0,C 180,E1 -20969.997,E2 -20969.997} C_VEL
LIN {X 0,Y 204.593,Z 465.179,A -85,B 0,C 180,E1 -20971.965,E2 -20971.965} C_VEL
LIN {X 0,Y 204.532,Z 462.779,A -85,B 0,C 180,E1 -20974.801,E2 -20974.801} C_VEL
LIN {X 0,Y 204.676,Z 459.066,A -85,B 0,C 180,E1 -20977.89,E2 -20977.89} C_VEL
LIN {X 0,Y 205.118,Z 454.341,A -85,B 0,C 180,E1 -20980.858,E2 -20980.858} C_VEL
LIN {X 0,Y 206.211,Z 447.204,A -85,B 0,C 180,E1 -20984.301,E2 -20984.301} C_VEL
LIN {X 0,Y 207.656,Z 439.445,A -85,B 0,C 180,E1 -20987.221,E2 -20987.221} C_VEL
LIN {X 0,Y 208.864,Z 433.173,A -85,B 0,C 180,E1 -20989.147,E2 -20989.147} C_VEL
LIN {X 0,Y 210.824,Z 423.895,A -85,B 0,C 180,E1 -20991.506,E2 -20991.506} C_VEL
LIN {X 0,Y 212.647,Z 413.501,A -85,B 0,C 180,E1 -20993.618,E2 -20993.618} C_VEL
LIN {X 0,Y 214.71,Z 402.001,A -85,B 0,C 180,E1 -20995.437,E2 -20995.437} C_VEL
LIN {X 0,Y 216.293,Z 392.048,A -85,B 0,C 180,E1 -20996.661,E2 -20996.661} C_VEL
LIN {X 0,Y 217.817,Z 380.385,A -85,B 0,C 180,E1 -20997.758,E2 -20997.758} C_VEL
LIN {X 0,Y 219.004,Z 368.069,A -85,B 0,C 180,E1 -20998.571,E2 -20998.571} C_VEL
LIN {X 0,Y 219.777,Z 353.209,A -85,B 0,C 180,E1 -20999.151,E2 -20999.151} C_VEL
LIN {X 0,Y 221.166,Z 311.717,A -85,B 0,C 180,E1 -21000.463,E2 -21000.463} C_VEL
LIN {X 0,Y 217.188,Z 275.455,A -85,B 0,C 180,E1 -21002.265,E2 -21002.265} C_VEL
LIN {X 0,Y 211.454,Z 260.266,A -85,B 0,C 180,E1 -21003.609,E2 -21003.609} C_VEL
LIN {X 0,Y 209.053,Z 254.106,A -85,B 0,C 180,E1 -21004.232,E2 -21004.232} C_VEL
LIN {X 0,Y 207.188,Z 245.741,A -85,B 0,C 180,E1 -21007.964,E2 -21007.964} C_VEL
LIN {X 0,Y 206.685,Z 243.743,A -85,B 0,C 180,E1 -21008.97,E2 -21008.97} C_VEL
LIN {X 0,Y 206.612,Z 243.747,A -85,B 0,C 180,E1 -21012.858,E2 -21012.858} C_VEL
LIN {X 0,Y 206.676,Z 243.74,A -85,B 0,C 180,E1 -21017.148,E2 -21017.148} C_VEL
LIN {X 0,Y 206.74,Z 243.732,A -85,B 0,C 180,E1 -21021.42,E2 -21021.42} C_VEL
LIN {X 0,Y 206.678,Z 243.738,A -85,B 0,C 180,E1 -21024.684,E2 -21024.684} C_VEL
LIN {X 0,Y 206.691,Z 243.738,A -85,B 0,C 180,E1 -21029.333,E2 -21029.333} C_VEL
LIN {X 0,Y 206.71,Z 243.736,A -85,B 0,C 180,E1 -21033.768,E2 -21033.768} C_VEL
LIN {X 0,Y 206.757,Z 243.73,A -85,B 0,C 180,E1 -21038.043,E2 -21038.043} C_VEL
LIN {X 0,Y 206.847,Z 243.713,A -85,B 0,C 180,E1 -21042.194,E2 -21042.194} C_VEL
LIN {X 0,Y 206.852,Z 243.716,A -85,B 0,C 180,E1 -21046.241,E2 -21046.241} C_VEL
LIN {X 0,Y 207.074,Z 243.687,A -85,B 0,C 180,E1 -21050.229,E2 -21050.229} C_VEL
LIN {X 0,Y 207.134,Z 243.682,A -85,B 0,C 180,E1 -21052.199,E2 -21052.199} C_VEL
LIN {X 0,Y 207.344,Z 243.624,A -85,B 0,C 180,E1 -21058.057,E2 -21058.057} C_VEL
LIN {X 0,Y 207.473,Z 243.599,A -85,B 0,C 180,E1 -21059.999,E2 -21059.999} C_VEL
LIN {X 0,Y 207.036,Z 243.685,A -85,B 0,C 180,E1 -21063.892,E2 -21063.892} C_VEL
LIN {X 0,Y 207.097,Z 243.686,A -85,B 0,C 180,E1 -21067.801,E2 -21067.801} C_VEL
LIN {X 0,Y 206.881,Z 243.705,A -85,B 0,C 180,E1 -21071.76,E2 -21071.76} C_VEL
LIN {X 0,Y 206.791,Z 243.725,A -85,B 0,C 180,E1 -21075.776,E2 -21075.776} C_VEL
LIN {X 0,Y 206.683,Z 243.728,A -85,B 0,C 180,E1 -21079.879,E2 -21079.879} C_VEL
LIN {X 0,Y 206.708,Z 243.735,A -85,B 0,C 180,E1 -21084.078,E2 -21084.078} C_VEL
LIN {X 0,Y 206.665,Z 243.716,A -85,B 0,C 180,E1 -21088.43,E2 -21088.43} C_VEL
LIN {X 0,Y 206.669,Z 243.718,A -85,B 0,C 180,E1 -21092.962,E2 -21092.962} C_VEL
LIN {X 0,Y 206.65,Z 243.742,A -85,B 0,C 180,E1 -21097.745,E2 -21097.745} C_VEL
LIN {X 0,Y 206.614,Z 243.728,A -85,B 0,C 180,E1 -21101.565,E2 -21101.565} C_VEL
LIN {X 0,Y 206.611,Z 243.74,A -85,B 0,C 180,E1 -21105.587,E2 -21105.587} C_VEL
LIN {X 0,Y 206.634,Z 243.744,A -85,B 0,C 180,E1 -21109.751,E2 -21109.751} C_VEL
LIN {X 0,Y 206.684,Z 243.736,A -85,B 0,C 180,E1 -21114.694,E2 -21114.694} C_VEL
LIN {X 0,Y 206.694,Z 243.727,A -85,B 0,C 180,E1 -21119.341,E2 -21119.341} C_VEL
LIN {X 0,Y 206.72,Z 243.735,A -85,B 0,C 180,E1 -21123.777,E2 -21123.777} C_VEL
LIN {X 0,Y 206.724,Z 243.735,A -85,B 0,C 180,E1 -21128.045,E2 -21128.045} C_VEL
LIN {X 0,Y 206.768,Z 243.731,A -85,B 0,C 180,E1 -21130.787,E2 -21130.787} C_VEL
LIN {X 0,Y 207.777,Z 246.577,A -85,B 0,C 180,E1 -21131.062,E2 -21131.062} C_VEL
LIN {X 0,Y 214.139,Z 258.952,A -85,B 0,C 180,E1 -21132.45,E2 -21132.45} C_VEL
LIN {X 0,Y 220.803,Z 274.269,A -85,B 0,C 180,E1 -21133.891,E2 -21133.891} C_VEL
LIN {X 0,Y 222.283,Z 278.751,A -85,B 0,C 180,E1 -21134.235,E2 -21134.235} C_VEL
LIN {X 0,Y 219.611,Z 345.324,A -85,B 0,C 180,E1 -21136.344,E2 -21136.344} C_VEL
LIN {X 0,Y 218.649,Z 359.175,A -85,B 0,C 180,E1 -21137.179,E2 -21137.179} C_VEL
LIN {X 0,Y 217.306,Z 372.044,A -85,B 0,C 180,E1 -21138.343,E2 -21138.343} C_VEL
LIN {X 0,Y 215.583,Z 384.592,A -85,B 0,C 180,E1 -21139.913,E2 -21139.913} C_VEL
LIN {X 0,Y 213.829,Z 395.763,A -85,B 0,C 180,E1 -21141.737,E2 -21141.737} C_VEL
LIN {X 0,Y 211.841,Z 406.11,A -85,B 0,C 180,E1 -21143.878,E2 -21143.878} C_VEL
LIN {X 0,Y 210.029,Z 414.968,A -85,B 0,C 180,E1 -21146.166,E2 -21146.166} C_VEL
LIN {X 0,Y 208.214,Z 423.857,A -85,B 0,C 180,E1 -21149.036,E2 -21149.036} C_VEL
LIN {X 0,Y 206.766,Z 430.975,A -85,B 0,C 180,E1 -21151.951,E2 -21151.951} C_VEL
LIN {X 0,Y 205.739,Z 436.651,A -85,B 0,C 180,E1 -21154.902,E2 -21154.902} C_VEL
LIN {X 0,Y 205.002,Z 441.127,A -85,B 0,C 180,E1 -21157.885,E2 -21157.885} C_VEL
LIN {X 0,Y 204.623,Z 443.506,A -85,B 0,C 180,E1 -21159.891,E2 -21159.891} C_VEL
LIN {X 0,Y 204.355,Z 445.45,A -85,B 0,C 180,E1 -21161.911,E2 -21161.911} C_VEL
LIN {X 0,Y 204.3,Z 447.79,A -85,B 0,C 180,E1 -21165.592,E2 -21165.592} C_VEL
LIN {X 0,Y 204.46,Z 448.597,A -85,B 0,C 180,E1 -21168.023,E2 -21168.023} C_VEL
LIN {X 0,Y 204.798,Z 448.809,A -85,B 0,C 180,E1 -21170.072,E2 -21170.072} C_VEL
LIN {X 0,Y 205.445,Z 448.483,A -85,B 0,C 180,E1 -21172.538,E2 -21172.538} C_VEL
LIN {X 0,Y 206.835,Z 446.88,A -85,B 0,C 180,E1 -21176.215,E2 -21176.215} C_VEL
LIN {X 0,Y 208.172,Z 444.982,A -85,B 0,C 180,E1 -21178.626,E2 -21178.626} C_VEL
LIN {X 0,Y 210.693,Z 440.851,A -85,B 0,C 180,E1 -21182.257,E2 -21182.257} C_VEL
LIN {X 0,Y 213.343,Z 436.072,A -85,B 0,C 180,E1 -21185.204,E2 -21185.204} C_VEL
LIN {X 0,Y 216.52,Z 429.925,A -85,B 0,C 180,E1 -21188.077,E2 -21188.077} C_VEL
LIN {X 0,Y 220.176,Z 422.175,A -85,B 0,C 180,E1 -21190.871,E2 -21190.871} C_VEL
LIN {X 0,Y 223.538,Z 414.163,A -85,B 0,C 180,E1 -21193.142,E2 -21193.142} C_VEL
LIN {X 0,Y 226.903,Z 405.293,A -85,B 0,C 180,E1 -21195.132,E2 -21195.132} C_VEL
LIN {X 0,Y 230.512,Z 394.482,A -85,B 0,C 180,E1 -21197.03,E2 -21197.03} C_VEL
LIN {X 0,Y 233.503,Z 383.593,A -85,B 0,C 180,E1 -21198.536,E2 -21198.536} C_VEL
LIN {X 0,Y 235.923,Z 372.311,A -85,B 0,C 180,E1 -21199.759,E2 -21199.759} C_VEL
LIN {X 0,Y 238.071,Z 359.49,A -85,B 0,C 180,E1 -21200.752,E2 -21200.752} C_VEL
LIN {X 0,Y 239.473,Z 347.07,A -85,B 0,C 180,E1 -21201.41,E2 -21201.41} C_VEL
LIN {X 0,Y 241.635,Z 310.65,A -85,B 0,C 180,E1 -21202.492,E2 -21202.492} C_VEL
LIN {X 0,Y 242.26,Z 298.559,A -85,B 0,C 180,E1 -21202.846,E2 -21202.846} C_VEL
LIN {X 0,Y 236.955,Z 287.702,A -85,B 0,C 180,E1 -21204.566,E2 -21204.566} C_VEL
LIN {X 0,Y 230.039,Z 276.263,A -85,B 0,C 180,E1 -21206.9,E2 -21206.9} C_VEL
LIN {X 0,Y 223.798,Z 267.068,A -85,B 0,C 180,E1 -21209.186,E2 -21209.186} C_VEL
LIN {X 0,Y 220.285,Z 262.318,A -85,B 0,C 180,E1 -21210.564,E2 -21210.564} C_VEL
LIN {X 0,Y 217.501,Z 258.443,A -85,B 0,C 180,E1 -21211.734,E2 -21211.734} C_VEL
LIN {X 0,Y 215,Z 255.01,A -85,B 0,C 180,E1 -21212.837,E2 -21212.837} C_VEL
LIN {X 0,Y 213.666,Z 253.527,A -85,B 0,C 180,E1 -21213.428,E2 -21213.428} C_VEL
LIN {X 0,Y 211.461,Z 250.65,A -85,B 0,C 180,E1 -21214.468,E2 -21214.468} C_VEL
LIN {X 0,Y 210.759,Z 249.251,A -85,B 0,C 180,E1 -21214.84,E2 -21214.84} C_VEL
LIN {X 0,Y 208.426,Z 247.506,A -85,B 0,C 180,E1 -21215.934,E2 -21215.934} C_VEL
LIN {X 0,Y 207.173,Z 245.29,A -85,B 0,C 180,E1 -21216.631,E2 -21216.631} C_VEL
LIN {X 0,Y 206.814,Z 243.721,A -85,B 0,C 180,E1 -21216.961,E2 -21216.961} C_VEL
LIN {X 0,Y 206.865,Z 243.706,A -85,B 0,C 180,E1 -21222.196,E2 -21222.196} C_VEL
LIN {X 0,Y 206.876,Z 243.708,A -85,B 0,C 180,E1 -21226.244,E2 -21226.244} C_VEL
LIN {X 0,Y 207.065,Z 243.689,A -85,B 0,C 180,E1 -21230.23,E2 -21230.23} C_VEL
LIN {X 0,Y 207.043,Z 243.692,A -85,B 0,C 180,E1 -21234.156,E2 -21234.156} C_VEL
LIN {X 0,Y 207.365,Z 243.644,A -85,B 0,C 180,E1 -21238.058,E2 -21238.058} C_VEL
LIN {X 0,Y 207.494,Z 243.623,A -85,B 0,C 180,E1 -21240.001,E2 -21240.001} C_VEL
LIN {X 0,Y 207.053,Z 243.685,A -85,B 0,C 180,E1 -21243.893,E2 -21243.893} C_VEL
LIN {X 0,Y 207.112,Z 243.679,A -85,B 0,C 180,E1 -21247.802,E2 -21247.802} C_VEL
LIN {X 0,Y 206.899,Z 243.7,A -85,B 0,C 180,E1 -21251.76,E2 -21251.76} C_VEL
LIN {X 0,Y 206.804,Z 243.711,A -85,B 0,C 180,E1 -21255.776,E2 -21255.776} C_VEL
LIN {X 0,Y 206.705,Z 243.724,A -85,B 0,C 180,E1 -21259.878,E2 -21259.878} C_VEL
LIN {X 0,Y 206.727,Z 243.724,A -85,B 0,C 180,E1 -21264.077,E2 -21264.077} C_VEL
LIN {X 0,Y 206.68,Z 243.734,A -85,B 0,C 180,E1 -21268.429,E2 -21268.429} C_VEL
LIN {X 0,Y 206.689,Z 243.753,A -85,B 0,C 180,E1 -21273.105,E2 -21273.105} C_VEL
LIN {X 0,Y 208.434,Z 248.819,A -85,B 0,C 180,E1 -21277.368,E2 -21277.368} C_VEL
LIN {X 0,Y 209.108,Z 251.107,A -85,B 0,C 180,E1 -21279.004,E2 -21279.004} C_VEL
LIN {X 0,Y 212.062,Z 255.702,A -85,B 0,C 180,E1 -21280.493,E2 -21280.493} C_VEL
LIN {X 0,Y 213.782,Z 257.949,A -85,B 0,C 180,E1 -21281.291,E2 -21281.291} C_VEL
LIN {X 0,Y 217.158,Z 263.022,A -85,B 0,C 180,E1 -21282.816,E2 -21282.816} C_VEL
LIN {X 0,Y 217.746,Z 263.991,A -85,B 0,C 180,E1 -21283.076,E2 -21283.076} C_VEL
LIN {X 0,Y 218.997,Z 268.505,A -85,B 0,C 180,E1 -21283.75,E2 -21283.75} C_VEL
LIN {X 0,Y 220.996,Z 279.437,A -85,B 0,C 180,E1 -21284.976,E2 -21284.976} C_VEL
LIN {X 0,Y 222.21,Z 282.588,A -85,B 0,C 180,E1 -21285.518,E2 -21285.518} C_VEL
LIN {X 0,Y 227.779,Z 293.246,A -85,B 0,C 180,E1 -21287.681,E2 -21287.681} C_VEL
LIN {X 0,Y 234.038,Z 307.275,A -85,B 0,C 180,E1 -21289.974,E2 -21289.974} C_VEL
LIN {X 0,Y 234.899,Z 310.052,A -85,B 0,C 180,E1 -21290.309,E2 -21290.309} C_VEL
LIN {X 0,Y 236.07,Z 320.842,A -85,B 0,C 180,E1 -21291.056,E2 -21291.056} C_VEL
LIN {X 0,Y 233.521,Z 362.818,A -85,B 0,C 180,E1 -21292.308,E2 -21292.308} C_VEL
LIN {X 0,Y 231.703,Z 376.447,A -85,B 0,C 180,E1 -21292.994,E2 -21292.994} C_VEL
LIN {X 0,Y 229.188,Z 389.214,A -85,B 0,C 180,E1 -21293.958,E2 -21293.958} C_VEL
LIN {X 0,Y 226.14,Z 400.902,A -85,B 0,C 180,E1 -21295.176,E2 -21295.176} C_VEL
LIN {X 0,Y 222.574,Z 412.194,A -85,B 0,C 180,E1 -21296.726,E2 -21296.726} C_VEL
LIN {X 0,Y 218.807,Z 422.41,A -85,B 0,C 180,E1 -21298.537,E2 -21298.537} C_VEL
LIN {X 0,Y 215.022,Z 431.61,A -85,B 0,C 180,E1 -21300.641,E2 -21300.641} C_VEL
LIN {X 0,Y 210.888,Z 440.581,A -85,B 0,C 180,E1 -21303.262,E2 -21303.262} C_VEL
LIN {X 0,Y 207.408,Z 447.838,A -85,B 0,C 180,E1 -21306.006,E2 -21306.006} C_VEL
LIN {X 0,Y 204.449,Z 453.688,A -85,B 0,C 180,E1 -21308.84,E2 -21308.84} C_VEL
LIN {X 0,Y 201.942,Z 458.329,A -85,B 0,C 180,E1 -21311.745,E2 -21311.745} C_VEL
LIN {X 0,Y 199.902,Z 461.892,A -85,B 0,C 180,E1 -21314.709,E2 -21314.709} C_VEL
LIN {X 0,Y 198.56,Z 464.482,A -85,B 0,C 180,E1 -21317.736,E2 -21317.736} C_VEL
LIN {X 0,Y 197.963,Z 465.723,A -85,B 0,C 180,E1 -21319.773,E2 -21319.773} C_VEL
LIN {X 0,Y 197.344,Z 466.959,A -85,B 0,C 180,E1 -21323.864,E2 -21323.864} C_VEL
LIN {X 0,Y 197.357,Z 467.007,A -85,B 0,C 180,E1 -21325.913,E2 -21325.913} C_VEL
LIN {X 0,Y 197.479,Z 466.672,A -85,B 0,C 180,E1 -21327.957,E2 -21327.957} C_VEL
LIN {X 0,Y 197.612,Z 465.916,A -85,B 0,C 180,E1 -21329.996,E2 -21329.996} C_VEL
LIN {X 0,Y 197.506,Z 464.708,A -85,B 0,C 180,E1 -21332.036,E2 -21332.036} C_VEL
LIN {X 0,Y 197.433,Z 462.583,A -85,B 0,C 180,E1 -21334.641,E2 -21334.641} C_VEL
LIN {X 0,Y 197.631,Z 458.455,A -85,B 0,C 180,E1 -21338.173,E2 -21338.173} C_VEL
LIN {X 0,Y 198.111,Z 453.651,A -85,B 0,C 180,E1 -21341.247,E2 -21341.247} C_VEL
LIN {X 0,Y 199.061,Z 447.559,A -85,B 0,C 180,E1 -21344.303,E2 -21344.303} C_VEL
LIN {X 0,Y 200.532,Z 439.96,A -85,B 0,C 180,E1 -21347.326,E2 -21347.326} C_VEL
LIN {X 0,Y 201.953,Z 432.89,A -85,B 0,C 180,E1 -21349.602,E2 -21349.602} C_VEL
LIN {X 0,Y 203.971,Z 423.771,A -85,B 0,C 180,E1 -21352,E2 -21352} C_VEL
LIN {X 0,Y 205.861,Z 413.434,A -85,B 0,C 180,E1 -21354.178,E2 -21354.178} C_VEL
LIN {X 0,Y 208.007,Z 401.995,A -85,B 0,C 180,E1 -21356.049,E2 -21356.049} C_VEL
LIN {X 0,Y 209.626,Z 392.118,A -85,B 0,C 180,E1 -21357.309,E2 -21357.309} C_VEL
LIN {X 0,Y 211.199,Z 380.575,A -85,B 0,C 180,E1 -21358.436,E2 -21358.436} C_VEL
LIN {X 0,Y 212.492,Z 367.498,A -85,B 0,C 180,E1 -21359.328,E2 -21359.328} C_VEL
LIN {X 0,Y 213.331,Z 351.428,A -85,B 0,C 180,E1 -21359.958,E2 -21359.958} C_VEL
LIN {X 0,Y 214.683,Z 312.028,A -85,B 0,C 180,E1 -21361.24,E2 -21361.24} C_VEL
LIN {X 0,Y 211.05,Z 277.753,A -85,B 0,C 180,E1 -21363.002,E2 -21363.002} C_VEL
LIN {X 0,Y 204.69,Z 260.959,A -85,B 0,C 180,E1 -21364.571,E2 -21364.571} C_VEL
LIN {X 0,Y 201.799,Z 253.752,A -85,B 0,C 180,E1 -21365.343,E2 -21365.343} C_VEL
LIN {X 0,Y 199.638,Z 244.62,A -85,B 0,C 180,E1 -21369.695,E2 -21369.695} C_VEL
LIN {X 0,Y 199.599,Z 244.62,A -85,B 0,C 180,E1 -21375.233,E2 -21375.233} C_VEL
LIN {X 0,Y 199.637,Z 244.617,A -85,B 0,C 180,E1 -21378.019,E2 -21378.019} C_VEL
LIN {X 0,Y 199.661,Z 244.612,A -85,B 0,C 180,E1 -21380.738,E2 -21380.738} C_VEL
LIN {X 0,Y 199.591,Z 244.622,A -85,B 0,C 180,E1 -21385.708,E2 -21385.708} C_VEL
LIN {X 0,Y 199.67,Z 244.612,A -85,B 0,C 180,E1 -21388.131,E2 -21388.131} C_VEL
LIN {X 0,Y 199.663,Z 244.612,A -85,B 0,C 180,E1 -21392.768,E2 -21392.768} C_VEL
LIN {X 0,Y 199.727,Z 244.603,A -85,B 0,C 180,E1 -21397.227,E2 -21397.227} C_VEL
LIN {X 0,Y 199.811,Z 244.588,A -85,B 0,C 180,E1 -21401.719,E2 -21401.719} C_VEL
LIN {X 0,Y 199.794,Z 244.596,A -85,B 0,C 180,E1 -21405.745,E2 -21405.745} C_VEL
LIN {X 0,Y 200.042,Z 244.563,A -85,B 0,C 180,E1 -21409.882,E2 -21409.882} C_VEL
LIN {X 0,Y 199.998,Z 244.567,A -85,B 0,C 180,E1 -21413.948,E2 -21413.948} C_VEL
LIN {X 0,Y 200.284,Z 244.502,A -85,B 0,C 180,E1 -21417.988,E2 -21417.988} C_VEL
LIN {X 0,Y 200.438,Z 244.473,A -85,B 0,C 180,E1 -21419.999,E2 -21419.999} C_VEL
LIN {X 0,Y 199.981,Z 244.564,A -85,B 0,C 180,E1 -21424.03,E2 -21424.03} C_VEL
LIN {X 0,Y 200.044,Z 244.564,A -85,B 0,C 180,E1 -21428.078,E2 -21428.078} C_VEL
LIN {X 0,Y 199.832,Z 244.583,A -85,B 0,C 180,E1 -21432.181,E2 -21432.181} C_VEL
LIN {X 0,Y 199.724,Z 244.606,A -85,B 0,C 180,E1 -21436.35,E2 -21436.35} C_VEL
LIN {X 0,Y 199.616,Z 244.611,A -85,B 0,C 180,E1 -21440.614,E2 -21440.614} C_VEL
LIN {X 0,Y 199.627,Z 244.614,A -85,B 0,C 180,E1 -21444.99,E2 -21444.99} C_VEL
LIN {X 0,Y 199.584,Z 244.588,A -85,B 0,C 180,E1 -21449.536,E2 -21449.536} C_VEL
LIN {X 0,Y 199.639,Z 244.587,A -85,B 0,C 180,E1 -21452.355,E2 -21452.355} C_VEL
LIN {X 0,Y 199.596,Z 244.622,A -85,B 0,C 180,E1 -21456.768,E2 -21456.768} C_VEL
LIN {X 0,Y 199.575,Z 244.619,A -85,B 0,C 180,E1 -21459.335,E2 -21459.335} C_VEL
LIN {X 0,Y 199.548,Z 244.601,A -85,B 0,C 180,E1 -21462.313,E2 -21462.313} C_VEL
LIN {X 0,Y 199.557,Z 244.615,A -85,B 0,C 180,E1 -21465.232,E2 -21465.232} C_VEL
LIN {X 0,Y 199.556,Z 244.628,A -85,B 0,C 180,E1 -21468.008,E2 -21468.008} C_VEL
LIN {X 0,Y 199.583,Z 244.614,A -85,B 0,C 180,E1 -21470.777,E2 -21470.777} C_VEL
LIN {X 0,Y 199.598,Z 244.621,A -85,B 0,C 180,E1 -21475.718,E2 -21475.718} C_VEL
LIN {X 0,Y 199.68,Z 244.605,A -85,B 0,C 180,E1 -21478.141,E2 -21478.141} C_VEL
LIN {X 0,Y 199.674,Z 244.613,A -85,B 0,C 180,E1 -21482.777,E2 -21482.777} C_VEL
LIN {X 0,Y 199.703,Z 244.609,A -85,B 0,C 180,E1 -21487.231,E2 -21487.231} C_VEL
LIN {X 0,Y 199.67,Z 244.615,A -85,B 0,C 180,E1 -21489.686,E2 -21489.686} C_VEL
LIN {X 0,Y 200.676,Z 247.449,A -85,B 0,C 180,E1 -21489.992,E2 -21489.992} C_VEL
LIN {X 0,Y 207.083,Z 259.544,A -85,B 0,C 180,E1 -21491.465,E2 -21491.465} C_VEL
LIN {X 0,Y 213.894,Z 274.742,A -85,B 0,C 180,E1 -21493.009,E2 -21493.009} C_VEL
LIN {X 0,Y 215.848,Z 280.176,A -85,B 0,C 180,E1 -21493.471,E2 -21493.471} C_VEL
LIN {X 0,Y 213.152,Z 344.93,A -85,B 0,C 180,E1 -21495.563,E2 -21495.563} C_VEL
LIN {X 0,Y 212.212,Z 358.333,A -85,B 0,C 180,E1 -21496.368,E2 -21496.368} C_VEL
LIN {X 0,Y 210.883,Z 370.906,A -85,B 0,C 180,E1 -21497.494,E2 -21497.494} C_VEL
LIN {X 0,Y 209.332,Z 382.245,A -85,B 0,C 180,E1 -21498.874,E2 -21498.874} C_VEL
LIN {X 0,Y 207.422,Z 393.92,A -85,B 0,C 180,E1 -21500.743,E2 -21500.743} C_VEL
LIN {X 0,Y 205.335,Z 405.02,A -85,B 0,C 180,E1 -21503.013,E2 -21503.013} C_VEL
LIN {X 0,Y 203.276,Z 414.728,A -85,B 0,C 180,E1 -21505.542,E2 -21505.542} C_VEL
LIN {X 0,Y 201.332,Z 423.716,A -85,B 0,C 180,E1 -21508.503,E2 -21508.503} C_VEL
LIN {X 0,Y 199.808,Z 430.946,A -85,B 0,C 180,E1 -21511.515,E2 -21511.515} C_VEL
LIN {X 0,Y 198.863,Z 435.824,A -85,B 0,C 180,E1 -21514.056,E2 -21514.056} C_VEL
LIN {X 0,Y 198.176,Z 440.087,A -85,B 0,C 180,E1 -21516.801,E2 -21516.801} C_VEL
LIN {X 0,Y 197.478,Z 444.197,A -85,B 0,C 180,E1 -21520.253,E2 -21520.253} C_VEL
LIN {X 0,Y 197.227,Z 446.041,A -85,B 0,C 180,E1 -21522.348,E2 -21522.348} C_VEL
LIN {X 0,Y 197.225,Z 448.122,A -85,B 0,C 180,E1 -21525.821,E2 -21525.821} C_VEL
LIN {X 0,Y 197.444,Z 449.002,A -85,B 0,C 180,E1 -21528.686,E2 -21528.686} C_VEL
LIN {X 0,Y 197.863,Z 449.12,A -85,B 0,C 180,E1 -21530.807,E2 -21530.807} C_VEL
LIN {X 0,Y 198.471,Z 448.823,A -85,B 0,C 180,E1 -21532.976,E2 -21532.976} C_VEL
LIN {X 0,Y 199.198,Z 448.141,A -85,B 0,C 180,E1 -21535.049,E2 -21535.049} C_VEL
LIN {X 0,Y 200.173,Z 446.974,A -85,B 0,C 180,E1 -21537.158,E2 -21537.158} C_VEL
LIN {X 0,Y 202.036,Z 444.389,A -85,B 0,C 180,E1 -21540.292,E2 -21540.292} C_VEL
LIN {X 0,Y 204.402,Z 440.699,A -85,B 0,C 180,E1 -21543.377,E2 -21543.377} C_VEL
LIN {X 0,Y 207.274,Z 435.785,A -85,B 0,C 180,E1 -21546.397,E2 -21546.397} C_VEL
LIN {X 0,Y 210.696,Z 429.497,A -85,B 0,C 180,E1 -21549.328,E2 -21549.328} C_VEL
LIN {X 0,Y 214.58,Z 421.559,A -85,B 0,C 180,E1 -21552.177,E2 -21552.177} C_VEL
LIN {X 0,Y 218.155,Z 413.304,A -85,B 0,C 180,E1 -21554.482,E2 -21554.482} C_VEL
LIN {X 0,Y 221.65,Z 404.365,A -85,B 0,C 180,E1 -21556.461,E2 -21556.461} C_VEL
LIN {X 0,Y 225.475,Z 393.069,A -85,B 0,C 180,E1 -21558.422,E2 -21558.422} C_VEL
LIN {X 0,Y 228.496,Z 382.047,A -85,B 0,C 180,E1 -21559.902,E2 -21559.902} C_VEL
LIN {X 0,Y 230.954,Z 370.797,A -85,B 0,C 180,E1 -21561.065,E2 -21561.065} C_VEL
LIN {X 0,Y 233.147,Z 357.647,A -85,B 0,C 180,E1 -21562.046,E2 -21562.046} C_VEL
LIN {X 0,Y 234.374,Z 346.313,A -85,B 0,C 180,E1 -21562.623,E2 -21562.623} C_VEL
LIN {X 0,Y 237.08,Z 301.156,A -85,B 0,C 180,E1 -21563.956,E2 -21563.956} C_VEL
LIN {X 0,Y 232.591,Z 291.919,A -85,B 0,C 180,E1 -21565.491,E2 -21565.491} C_VEL
LIN {X 0,Y 225.539,Z 280.078,A -85,B 0,C 180,E1 -21568.013,E2 -21568.013} C_VEL
LIN {X 0,Y 219.566,Z 271.34,A -85,B 0,C 180,E1 -21570.327,E2 -21570.327} C_VEL
LIN {X 0,Y 214.383,Z 264.077,A -85,B 0,C 180,E1 -21572.549,E2 -21572.549} C_VEL
LIN {X 0,Y 211.285,Z 259.886,A -85,B 0,C 180,E1 -21573.983,E2 -21573.983} C_VEL
LIN {X 0,Y 208.704,Z 256.612,A -85,B 0,C 180,E1 -21575.24,E2 -21575.24} C_VEL
LIN {X 0,Y 207.879,Z 255.404,A -85,B 0,C 180,E1 -21575.668,E2 -21575.668} C_VEL
LIN {X 0,Y 205.367,Z 252.9,A -85,B 0,C 180,E1 -21576.947,E2 -21576.947} C_VEL
LIN {X 0,Y 203.84,Z 250.172,A -85,B 0,C 180,E1 -21577.846,E2 -21577.846} C_VEL
LIN {X 0,Y 201.317,Z 248.304,A -85,B 0,C 180,E1 -21579.234,E2 -21579.234} C_VEL
LIN {X 0,Y 200.094,Z 246.179,A -85,B 0,C 180,E1 -21580.041,E2 -21580.041} C_VEL
LIN {X 0,Y 199.716,Z 244.6,A -85,B 0,C 180,E1 -21580.404,E2 -21580.404} C_VEL
LIN {X 0,Y 199.79,Z 244.586,A -85,B 0,C 180,E1 -21583.656,E2 -21583.656} C_VEL
LIN {X 0,Y 199.86,Z 244.576,A -85,B 0,C 180,E1 -21587.82,E2 -21587.82} C_VEL
LIN {X 0,Y 200.068,Z 244.547,A -85,B 0,C 180,E1 -21591.923,E2 -21591.923} C_VEL
LIN {X 0,Y 200.305,Z 244.522,A -85,B 0,C 180,E1 -21597.99,E2 -21597.99} C_VEL
LIN {X 0,Y 200.459,Z 244.499,A -85,B 0,C 180,E1 -21600.001,E2 -21600.001} C_VEL
LIN {X 0,Y 199.998,Z 244.562,A -85,B 0,C 180,E1 -21604.031,E2 -21604.031} C_VEL
LIN {X 0,Y 200.061,Z 244.557,A -85,B 0,C 180,E1 -21608.078,E2 -21608.078} C_VEL
LIN {X 0,Y 199.85,Z 244.583,A -85,B 0,C 180,E1 -21612.182,E2 -21612.182} C_VEL
LIN {X 0,Y 199.741,Z 244.596,A -85,B 0,C 180,E1 -21616.349,E2 -21616.349} C_VEL
LIN {X 0,Y 199.639,Z 244.61,A -85,B 0,C 180,E1 -21620.613,E2 -21620.613} C_VEL
LIN {X 0,Y 199.642,Z 244.615,A -85,B 0,C 180,E1 -21624.989,E2 -21624.989} C_VEL
LIN {X 0,Y 199.625,Z 244.614,A -85,B 0,C 180,E1 -21629.967,E2 -21629.967} C_VEL
LIN {X 0,Y 200.954,Z 248.702,A -85,B 0,C 180,E1 -21634.027,E2 -21634.027} C_VEL
LIN {X 0,Y 201.713,Z 250.535,A -85,B 0,C 180,E1 -21635.551,E2 -21635.551} C_VEL
LIN {X 0,Y 204.204,Z 254.412,A -85,B 0,C 180,E1 -21637.035,E2 -21637.035} C_VEL
LIN {X 0,Y 206.702,Z 257.662,A -85,B 0,C 180,E1 -21638.385,E2 -21638.385} C_VEL
LIN {X 0,Y 209.989,Z 262.482,A -85,B 0,C 180,E1 -21640.073,E2 -21640.073} C_VEL
LIN {X 0,Y 215.234,Z 270.719,A -85,B 0,C 180,E1 -21642.556,E2 -21642.556} C_VEL
LIN {X 0,Y 218.499,Z 276.165,A -85,B 0,C 180,E1 -21643.991,E2 -21643.991} C_VEL
LIN {X 0,Y 222.21,Z 282.588,A -85,B 0,C 180,E1 -21645.518,E2 -21645.518} C_VEL
LIN {X 0,Y 224.055,Z 287.259,A -85,B 0,C 180,E1 -21646.313,E2 -21646.313} C_VEL
LIN {X 0,Y 225.972,Z 296.169,A -85,B 0,C 180,E1 -21647.307,E2 -21647.307} C_VEL
LIN {X 0,Y 228.155,Z 307.114,A -85,B 0,C 180,E1 -21648.432,E2 -21648.432} C_VEL
LIN {X 0,Y 229.293,Z 310.465,A -85,B 0,C 180,E1 -21648.894,E2 -21648.894} C_VEL
LIN {X 0,Y 230.081,Z 312.955,A -85,B 0,C 180,E1 -21649.215,E2 -21649.215} C_VEL
LIN {X 0,Y 231.025,Z 321.766,A -85,B 0,C 180,E1 -21649.853,E2 -21649.853} C_VEL
LIN {X 0,Y 228.433,Z 362.571,A -85,B 0,C 180,E1 -21651.086,E2 -21651.086} C_VEL
LIN {X 0,Y 226.511,Z 376.363,A -85,B 0,C 180,E1 -21651.786,E2 -21651.786} C_VEL
LIN {X 0,Y 224.047,Z 388.541,A -85,B 0,C 180,E1 -21652.714,E2 -21652.714} C_VEL
LIN {X 0,Y 220.878,Z 400.305,A -85,B 0,C 180,E1 -21653.939,E2 -21653.939} C_VEL
LIN {X 0,Y 217.145,Z 411.65,A -85,B 0,C 180,E1 -21655.501,E2 -21655.501} C_VEL
LIN {X 0,Y 213.213,Z 421.908,A -85,B 0,C 180,E1 -21657.332,E2 -21657.332} C_VEL
LIN {X 0,Y 208.872,Z 431.956,A -85,B 0,C 180,E1 -21659.687,E2 -21659.687} C_VEL
LIN {X 0,Y 204.583,Z 440.814,A -85,B 0,C 180,E1 -21662.369,E2 -21662.369} C_VEL
LIN {X 0,Y 200.931,Z 447.965,A -85,B 0,C 180,E1 -21665.181,E2 -21665.181} C_VEL
LIN {X 0,Y 197.842,Z 453.71,A -85,B 0,C 180,E1 -21668.098,E2 -21668.098} C_VEL
LIN {X 0,Y 195.174,Z 458.27,A -85,B 0,C 180,E1 -21671.088,E2 -21671.088} C_VEL
LIN {X 0,Y 193.037,Z 461.771,A -85,B 0,C 180,E1 -21674.152,E2 -21674.152} C_VEL
LIN {X 0,Y 191.603,Z 464.297,A -85,B 0,C 180,E1 -21677.284,E2 -21677.284} C_VEL
LIN {X 0,Y 190.961,Z 465.484,A -85,B 0,C 180,E1 -21679.393,E2 -21679.393} C_VEL
LIN {X 0,Y 190.279,Z 466.646,A -85,B 0,C 180,E1 -21683.635,E2 -21683.635} C_VEL
LIN {X 0,Y 190.279,Z 466.663,A -85,B 0,C 180,E1 -21685.76,E2 -21685.76} C_VEL
LIN {X 0,Y 190.392,Z 466.289,A -85,B 0,C 180,E1 -21687.881,E2 -21687.881} C_VEL
LIN {X 0,Y 190.547,Z 465.477,A -85,B 0,C 180,E1 -21689.996,E2 -21689.996} C_VEL
LIN {X 0,Y 190.421,Z 464.235,A -85,B 0,C 180,E1 -21692.111,E2 -21692.111} C_VEL
LIN {X 0,Y 190.337,Z 462.373,A -85,B 0,C 180,E1 -21694.47,E2 -21694.47} C_VEL
LIN {X 0,Y 190.486,Z 459.211,A -85,B 0,C 180,E1 -21697.415,E2 -21697.415} C_VEL
LIN {X 0,Y 190.87,Z 454.729,A -85,B 0,C 180,E1 -21700.604,E2 -21700.604} C_VEL
LIN {X 0,Y 191.706,Z 449.014,A -85,B 0,C 180,E1 -21703.781,E2 -21703.781} C_VEL
LIN {X 0,Y 193.206,Z 441.843,A -85,B 0,C 180,E1 -21706.913,E2 -21706.913} C_VEL
LIN {X 0,Y 194.911,Z 433.455,A -85,B 0,C 180,E1 -21709.826,E2 -21709.826} C_VEL
LIN {X 0,Y 196.672,Z 425.616,A -85,B 0,C 180,E1 -21712.032,E2 -21712.032} C_VEL
LIN {X 0,Y 198.672,Z 415.831,A -85,B 0,C 180,E1 -21714.276,E2 -21714.276} C_VEL
LIN {X 0,Y 200.8,Z 405.139,A -85,B 0,C 180,E1 -21716.217,E2 -21716.217} C_VEL
LIN {X 0,Y 202.852,Z 393.197,A -85,B 0,C 180,E1 -21717.88,E2 -21717.88} C_VEL
LIN {X 0,Y 204.612,Z 380.765,A -85,B 0,C 180,E1 -21719.157,E2 -21719.157} C_VEL
LIN {X 0,Y 205.946,Z 367.995,A -85,B 0,C 180,E1 -21720.074,E2 -21720.074} C_VEL
LIN {X 0,Y 206.822,Z 353.162,A -85,B 0,C 180,E1 -21720.694,E2 -21720.694} C_VEL
LIN {X 0,Y 208.3,Z 312.916,A -85,B 0,C 180,E1 -21722.035,E2 -21722.035} C_VEL
LIN {X 0,Y 204.818,Z 279.656,A -85,B 0,C 180,E1 -21723.816,E2 -21723.816} C_VEL
LIN {X 0,Y 198.857,Z 264.03,A -85,B 0,C 180,E1 -21725.358,E2 -21725.358} C_VEL
LIN {X 0,Y 194.502,Z 253.395,A -85,B 0,C 180,E1 -21726.558,E2 -21726.558} C_VEL
LIN {X 0,Y 192.561,Z 245.5,A -85,B 0,C 180,E1 -21730.586,E2 -21730.586} C_VEL
LIN {X 0,Y 192.535,Z 245.503,A -85,B 0,C 180,E1 -21736.088,E2 -21736.088} C_VEL
LIN {X 0,Y 192.569,Z 245.495,A -85,B 0,C 180,E1 -21740.021,E2 -21740.021} C_VEL
LIN {X 0,Y 192.566,Z 245.497,A -85,B 0,C 180,E1 -21744.271,E2 -21744.271} C_VEL
LIN {X 0,Y 192.577,Z 245.496,A -85,B 0,C 180,E1 -21749.274,E2 -21749.274} C_VEL
LIN {X 0,Y 192.641,Z 245.485,A -85,B 0,C 180,E1 -21751.687,E2 -21751.687} C_VEL
LIN {X 0,Y 192.688,Z 245.478,A -85,B 0,C 180,E1 -21756.346,E2 -21756.346} C_VEL
LIN {X 0,Y 192.756,Z 245.467,A -85,B 0,C 180,E1 -21761.41,E2 -21761.41} C_VEL
LIN {X 0,Y 192.724,Z 245.48,A -85,B 0,C 180,E1 -21765.21,E2 -21765.21} C_VEL
LIN {X 0,Y 192.953,Z 245.443,A -85,B 0,C 180,E1 -21769.506,E2 -21769.506} C_VEL
LIN {X 0,Y 193.03,Z 245.44,A -85,B 0,C 180,E1 -21771.625,E2 -21771.625} C_VEL
LIN {X 0,Y 193.226,Z 245.379,A -85,B 0,C 180,E1 -21777.915,E2 -21777.915} C_VEL
LIN {X 0,Y 193.403,Z 245.348,A -85,B 0,C 180,E1 -21779.999,E2 -21779.999} C_VEL
LIN {X 0,Y 192.927,Z 245.442,A -85,B 0,C 180,E1 -21784.177,E2 -21784.177} C_VEL
LIN {X 0,Y 192.995,Z 245.443,A -85,B 0,C 180,E1 -21788.375,E2 -21788.375} C_VEL
LIN {X 0,Y 192.758,Z 245.465,A -85,B 0,C 180,E1 -21792.636,E2 -21792.636} C_VEL
LIN {X 0,Y 192.681,Z 245.481,A -85,B 0,C 180,E1 -21796.965,E2 -21796.965} C_VEL
LIN {X 0,Y 192.552,Z 245.496,A -85,B 0,C 180,E1 -21801.406,E2 -21801.406} C_VEL
LIN {X 0,Y 192.609,Z 245.492,A -85,B 0,C 180,E1 -21804.208,E2 -21804.208} C_VEL
LIN {X 0,Y 192.567,Z 245.466,A -85,B 0,C 180,E1 -21808.864,E2 -21808.864} C_VEL
LIN {X 0,Y 192.57,Z 245.474,A -85,B 0,C 180,E1 -21813.191,E2 -21813.191} C_VEL
LIN {X 0,Y 192.521,Z 245.501,A -85,B 0,C 180,E1 -21818.358,E2 -21818.358} C_VEL
LIN {X 0,Y 192.466,Z 245.481,A -85,B 0,C 180,E1 -21823.098,E2 -21823.098} C_VEL
LIN {X 0,Y 192.469,Z 245.509,A -85,B 0,C 180,E1 -21826.911,E2 -21826.911} C_VEL
LIN {X 0,Y 192.527,Z 245.486,A -85,B 0,C 180,E1 -21831.651,E2 -21831.651} C_VEL
LIN {X 0,Y 192.583,Z 245.495,A -85,B 0,C 180,E1 -21836.819,E2 -21836.819} C_VEL
LIN {X 0,Y 192.649,Z 245.486,A -85,B 0,C 180,E1 -21841.696,E2 -21841.696} C_VEL
LIN {X 0,Y 192.651,Z 245.489,A -85,B 0,C 180,E1 -21847.484,E2 -21847.484} C_VEL
LIN {X 0,Y 192.61,Z 245.494,A -85,B 0,C 180,E1 -21848.535,E2 -21848.535} C_VEL
LIN {X 0,Y 193.68,Z 248.418,A -85,B 0,C 180,E1 -21848.857,E2 -21848.857} C_VEL
LIN {X 0,Y 200.406,Z 260.902,A -85,B 0,C 180,E1 -21850.499,E2 -21850.499} C_VEL
LIN {X 0,Y 207.367,Z 276.232,A -85,B 0,C 180,E1 -21852.157,E2 -21852.157} C_VEL
LIN {X 0,Y 209.525,Z 281.931,A -85,B 0,C 180,E1 -21852.682,E2 -21852.682} C_VEL
LIN {X 0,Y 206.663,Z 345.618,A -85,B 0,C 180,E1 -21854.787,E2 -21854.787} C_VEL
LIN {X 0,Y 205.63,Z 359.464,A -85,B 0,C 180,E1 -21855.658,E2 -21855.658} C_VEL
LIN {X 0,Y 204.243,Z 371.931,A -85,B 0,C 180,E1 -21856.827,E2 -21856.827} C_VEL
LIN {X 0,Y 202.645,Z 383.066,A -85,B 0,C 180,E1 -21858.248,E2 -21858.248} C_VEL
LIN {X 0,Y 200.647,Z 394.651,A -85,B 0,C 180,E1 -21860.173,E2 -21860.173} C_VEL
LIN {X 0,Y 198.473,Z 405.68,A -85,B 0,C 180,E1 -21862.515,E2 -21862.515} C_VEL
LIN {X 0,Y 196.527,Z 414.493,A -85,B 0,C 180,E1 -21864.875,E2 -21864.875} C_VEL
LIN {X 0,Y 194.479,Z 423.574,A -85,B 0,C 180,E1 -21867.933,E2 -21867.933} C_VEL
LIN {X 0,Y 192.889,Z 430.891,A -85,B 0,C 180,E1 -21871.047,E2 -21871.047} C_VEL
LIN {X 0,Y 191.705,Z 436.742,A -85,B 0,C 180,E1 -21874.208,E2 -21874.208} C_VEL
LIN {X 0,Y 190.939,Z 441.223,A -85,B 0,C 180,E1 -21877.306,E2 -21877.306} C_VEL
LIN {X 0,Y 190.312,Z 444.866,A -85,B 0,C 180,E1 -21880.643,E2 -21880.643} C_VEL
LIN {X 0,Y 190.119,Z 446.619,A -85,B 0,C 180,E1 -21882.817,E2 -21882.817} C_VEL
LIN {X 0,Y 190.142,Z 448.45,A -85,B 0,C 180,E1 -21886.055,E2 -21886.055} C_VEL
LIN {X 0,Y 190.479,Z 449.368,A -85,B 0,C 180,E1 -21889.396,E2 -21889.396} C_VEL
LIN {X 0,Y 191.523,Z 449.16,A -85,B 0,C 180,E1 -21893.455,E2 -21893.455} C_VEL
LIN {X 0,Y 192.483,Z 448.307,A -85,B 0,C 180,E1 -21895.987,E2 -21895.987} C_VEL
LIN {X 0,Y 194.627,Z 445.727,A -85,B 0,C 180,E1 -21899.93,E2 -21899.93} C_VEL
LIN {X 0,Y 197.284,Z 441.97,A -85,B 0,C 180,E1 -21903.517,E2 -21903.517} C_VEL
LIN {X 0,Y 200.213,Z 437.364,A -85,B 0,C 180,E1 -21906.638,E2 -21906.638} C_VEL
LIN {X 0,Y 203.683,Z 431.394,A -85,B 0,C 180,E1 -21909.668,E2 -21909.668} C_VEL
LIN {X 0,Y 207.662,Z 423.825,A -85,B 0,C 180,E1 -21912.599,E2 -21912.599} C_VEL
LIN {X 0,Y 211.311,Z 416.066,A -85,B 0,C 180,E1 -21914.957,E2 -21914.957} C_VEL
LIN {X 0,Y 214.918,Z 407.513,A -85,B 0,C 180,E1 -21917.027,E2 -21917.027} C_VEL
LIN {X 0,Y 218.83,Z 397.062,A -85,B 0,C 180,E1 -21919.001,E2 -21919.001} C_VEL
LIN {X 0,Y 222.139,Z 386.288,A -85,B 0,C 180,E1 -21920.593,E2 -21920.593} C_VEL
LIN {X 0,Y 225.139,Z 373.883,A -85,B 0,C 180,E1 -21922.017,E2 -21922.017} C_VEL
LIN {X 0,Y 227.527,Z 361.106,A -85,B 0,C 180,E1 -21923.056,E2 -21923.056} C_VEL
LIN {X 0,Y 229.122,Z 348.243,A -85,B 0,C 180,E1 -21923.77,E2 -21923.77} C_VEL
LIN {X 0,Y 230.787,Z 324.513,A -85,B 0,C 180,E1 -21924.5,E2 -21924.5} C_VEL
LIN {X 0,Y 231.925,Z 303.609,A -85,B 0,C 180,E1 -21925.14,E2 -21925.14} C_VEL
LIN {X 0,Y 228.122,Z 295.818,A -85,B 0,C 180,E1 -21926.52,E2 -21926.52} C_VEL
LIN {X 0,Y 221.597,Z 284.789,A -85,B 0,C 180,E1 -21928.978,E2 -21928.978} C_VEL
LIN {X 0,Y 215.021,Z 274.835,A -85,B 0,C 180,E1 -21931.711,E2 -21931.711} C_VEL
LIN {X 0,Y 211.27,Z 269.673,A -85,B 0,C 180,E1 -21933.408,E2 -21933.408} C_VEL
LIN {X 0,Y 208.071,Z 265.365,A -85,B 0,C 180,E1 -21934.96,E2 -21934.96} C_VEL
LIN {X 0,Y 205.278,Z 261.566,A -85,B 0,C 180,E1 -21936.414,E2 -21936.414} C_VEL
LIN {X 0,Y 202.631,Z 258.632,A -85,B 0,C 180,E1 -21937.841,E2 -21937.841} C_VEL
LIN {X 0,Y 201.319,Z 256.542,A -85,B 0,C 180,E1 -21938.632,E2 -21938.632} C_VEL
LIN {X 0,Y 198.645,Z 254.009,A -85,B 0,C 180,E1 -21940.226,E2 -21940.226} C_VEL
LIN {X 0,Y 197.152,Z 251.199,A -85,B 0,C 180,E1 -21941.288,E2 -21941.288} C_VEL
LIN {X 0,Y 194.511,Z 249.36,A -85,B 0,C 180,E1 -21943.037,E2 -21943.037} C_VEL
LIN {X 0,Y 193.044,Z 246.813,A -85,B 0,C 180,E1 -21944.223,E2 -21944.223} C_VEL
LIN {X 0,Y 192.74,Z 245.471,A -85,B 0,C 180,E1 -21944.604,E2 -21944.604} C_VEL
LIN {X 0,Y 192.94,Z 245.452,A -85,B 0,C 180,E1 -21949.567,E2 -21949.567} C_VEL
LIN {X 0,Y 192.968,Z 245.442,A -85,B 0,C 180,E1 -21953.728,E2 -21953.728} C_VEL
LIN {X 0,Y 193.247,Z 245.4,A -85,B 0,C 180,E1 -21957.916,E2 -21957.916} C_VEL
LIN {X 0,Y 193.424,Z 245.375,A -85,B 0,C 180,E1 -21960.001,E2 -21960.001} C_VEL
LIN {X 0,Y 192.944,Z 245.438,A -85,B 0,C 180,E1 -21964.178,E2 -21964.178} C_VEL
LIN {X 0,Y 193.013,Z 245.434,A -85,B 0,C 180,E1 -21968.375,E2 -21968.375} C_VEL
LIN {X 0,Y 192.772,Z 245.467,A -85,B 0,C 180,E1 -21972.636,E2 -21972.636} C_VEL
LIN {X 0,Y 192.69,Z 245.469,A -85,B 0,C 180,E1 -21978.509,E2 -21978.509} C_VEL
LIN {X 0,Y 192.629,Z 245.48,A -85,B 0,C 180,E1 -21984.204,E2 -21984.204} C_VEL
LIN {X 0,Y 192.585,Z 245.514,A -85,B 0,C 180,E1 -21986.555,E2 -21986.555} C_VEL
LIN {X 0,Y 194.003,Z 249.655,A -85,B 0,C 180,E1 -21991.08,E2 -21991.08} C_VEL
LIN {X 0,Y 198.136,Z 255.429,A -85,B 0,C 180,E1 -21994.022,E2 -21994.022} C_VEL
LIN {X 0,Y 199.458,Z 257.023,A -85,B 0,C 180,E1 -21994.86,E2 -21994.86} C_VEL
LIN {X 0,Y 204.163,Z 263.869,A -85,B 0,C 180,E1 -21997.653,E2 -21997.653} C_VEL
LIN {X 0,Y 208.22,Z 270.068,A -85,B 0,C 180,E1 -21999.815,E2 -21999.815} C_VEL
LIN {X 0,Y 212.117,Z 276.271,A -85,B 0,C 180,E1 -22001.723,E2 -22001.723} C_VEL
LIN {X 0,Y 217.231,Z 285.119,A -85,B 0,C 180,E1 -22004.041,E2 -22004.041} C_VEL
LIN {X 0,Y 222.281,Z 294.746,A -85,B 0,C 180,E1 -22006.148,E2 -22006.148} C_VEL
LIN {X 0,Y 226.96,Z 304.988,A -85,B 0,C 180,E1 -22008.004,E2 -22008.004} C_VEL
LIN {X 0,Y 229.293,Z 310.465,A -85,B 0,C 180,E1 -22008.894,E2 -22008.894} C_VEL
LIN {X 0,Y 230.082,Z 313.887,A -85,B 0,C 180,E1 -22009.258,E2 -22009.258} C_VEL
LIN {X 0,Y 230.108,Z 317.666,A -85,B 0,C 180,E1 -22009.435,E2 -22009.435} C_VEL
LIN {X 0,Y 229.171,Z 323.547,A -85,B 0,C 180,E1 -22009.456,E2 -22009.456} C_VEL
LIN {X 0,Y 225.457,Z 337.801,A -85,B 0,C 180,E1 -22009.122,E2 -22009.122} C_VEL
LIN {X 0,Y 224.889,Z 341.991,A -85,B 0,C 180,E1 -22009.163,E2 -22009.163} C_VEL
LIN {X 0,Y 223.269,Z 363.767,A -85,B 0,C 180,E1 -22009.86,E2 -22009.86} C_VEL
LIN {X 0,Y 221.287,Z 377.049,A -85,B 0,C 180,E1 -22010.566,E2 -22010.566} C_VEL
LIN {X 0,Y 218.73,Z 388.88,A -85,B 0,C 180,E1 -22011.498,E2 -22011.498} C_VEL
LIN {X 0,Y 215.213,Z 401.284,A -85,B 0,C 180,E1 -22012.833,E2 -22012.833} C_VEL
LIN {X 0,Y 211.375,Z 412.389,A -85,B 0,C 180,E1 -22014.418,E2 -22014.418} C_VEL
LIN {X 0,Y 206.881,Z 423.384,A -85,B 0,C 180,E1 -22016.493,E2 -22016.493} C_VEL
LIN {X 0,Y 202.794,Z 432.302,A -85,B 0,C 180,E1 -22018.678,E2 -22018.678} C_VEL
LIN {X 0,Y 198.339,Z 441.046,A -85,B 0,C 180,E1 -22021.42,E2 -22021.42} C_VEL
LIN {X 0,Y 194.496,Z 448.066,A -85,B 0,C 180,E1 -22024.302,E2 -22024.302} C_VEL
LIN {X 0,Y 191.251,Z 453.717,A -85,B 0,C 180,E1 -22027.302,E2 -22027.302} C_VEL
LIN {X 0,Y 188.433,Z 458.2,A -85,B 0,C 180,E1 -22030.384,E2 -22030.384} C_VEL
LIN {X 0,Y 186.88,Z 460.584,A -85,B 0,C 180,E1 -22032.489,E2 -22032.489} C_VEL
LIN {X 0,Y 185.559,Z 462.549,A -85,B 0,C 180,E1 -22034.623,E2 -22034.623} C_VEL
LIN {X 0,Y 184.646,Z 464.111,A -85,B 0,C 180,E1 -22036.796,E2 -22036.796} C_VEL
